# B&R Automation Studio project CControl_Gschneitner (part 3)

#### fbMathTrGutGew.st - Berechnungen des Trockengutes (spez. Gewicht, Wasserentzug, Gewicht Start, Gewicht Ende...)
```iecst
(********************************************************************
 * COPYRIGHT -- LASCO Heu- und Forsttechnik GmbH
 ********************************************************************
 * Library: LascoMath
 * Datei: fbMathTrGutGew.st
 * Autor: Rudolf Lachner
 * Erstellt: 5. März 2014
 ********************************************************************
 * Implementierung der Library LascoMath
 ********************************************************************)

(* Berechnungen des Trockengutes (spez. Gewicht, Wasserentzug, Gewicht Start, Gewicht Ende...) *)
FUNCTION_BLOCK fbMathTrGutGew

	IF (Freigabe = TRUE) THEN

		//Boxentrocknung**************************************************************************************************************************************************
		IF (Anlagentyp = FALSE) THEN

			//Spez. Gewicht des Trockengutes [kg/m³]
			//**************************************

			//Heu
			IF (Trocknungsgut = 0) AND (FeuchteBeiStart <> 0) AND (FeuchteBeiStart < 100) THEN
				TrockengutSpezGewicht		:= (0.0237 * FeuchteBeiStart * FeuchteBeiStart - 0.395 * FeuchteBeiStart + 60.5) * 1.1;
				//Fichte
			ELSIF (Trocknungsgut = 1) AND (FeuchteBeiStart <> 0) AND (FeuchteBeiStart < 100) THEN
				TrockengutSpezGewicht 		:= (0.0313 * FeuchteBeiStart * FeuchteBeiStart + 1.2245 * FeuchteBeiStart + 151.32);
				//Buche
			ELSIF (Trocknungsgut = 2) AND (FeuchteBeiStart <> 0) AND (FeuchteBeiStart < 100) THEN
				TrockengutSpezGewicht 		:= (0.0462 * FeuchteBeiStart * FeuchteBeiStart + 1.7883 * FeuchteBeiStart + 222.47);
				//Mais
			ELSIF (Trocknungsgut = 3) AND (FeuchteBeiStart <> 0) AND (FeuchteBeiStart < 100) THEN
				TrockengutSpezGewicht 		:= (730 + 476 * (FeuchteBeiStart / (100 - FeuchteBeiStart)));
				//Weizen
			ELSIF (Trocknungsgut = 4) AND (FeuchteBeiStart <> 0) AND (FeuchteBeiStart < 100) THEN
				TrockengutSpezGewicht 		:= (680 + 476 * (FeuchteBeiStart / (100 - FeuchteBeiStart)));
			ELSIF (Trocknungsgut = 5) AND (SpezGewichtUser <> 0) AND (FeuchteBeiStart <> 0) AND (FeuchteBeiStart < 100) THEN
				TrockengutSpezGewicht		:= ((SpezGewichtUser - 476) + 476 * (FeuchteBeiStart / (100 - FeuchteBeiStart)));
			ELSE
				TrockengutSpezGewicht		:= CONST_MATH_MAX_VALUE;
			END_IF

			//Trockengut Gewicht bei Trocknungsstart [kg]
			//*******************************************
			IF (TrockengutSpezGewicht <> 0) AND (TrockengutSpezGewicht < CONST_MATH_MAX_VALUE) AND (FuellhoeheTrockengut > 0) AND
				(Boxenflaeche > 0) THEN
				TrockengutGewichtStart		:= Boxenflaeche * FuellhoeheTrockengut * TrockengutSpezGewicht;
			ELSE
				TrockengutGewichtStart		:= 0;
			END_IF

			//Rundballentrocknung***************************************************************************************************************************************************
		ELSE

			//Trockengut Gewicht bei Trocknungsstart [kg]
			//*******************************************
			IF (GewichtProBallen > 0) AND (AnzahlBallen > 0) THEN
				TrockengutGewichtStart		:= GewichtProBallen * AnzahlBallen;
			ELSE
				TrockengutGewichtStart		:= 0;
			END_IF

		END_IF

		//Trockengut Gewicht Substanz [kg]
		//********************************
		IF (TrockengutGewichtStart <> 0) AND (FeuchteBeiStart > 0) THEN
			TrockengutGewichtSubstanz	:= TrockengutGewichtStart - (TrockengutGewichtStart * FeuchteBeiStart / 100);
		ELSE
			TrockengutGewichtSubstanz	:= 0;
		END_IF

		IF (TrockengutGewichtSubstanz < 0) THEN
			TrockengutGewichtSubstanz	:= 0;
		END_IF

		//Trockengut Gewicht Ende [kg]
		//****************************
		IF (TrockengutGewichtSubstanz <> 0) AND (FeuchteEnde > 0) THEN
			loc_TrockengutGewichtEnde	:= ((100 - FeuchteEnde) / 100);
			IF (loc_TrockengutGewichtEnde <> 0) THEN
				TrockengutGewichtEnde	:= TrockengutGewichtSubstanz / loc_TrockengutGewichtEnde;
			ELSE
				TrockengutGewichtEnde	:= 0;
			END_IF
		ELSE
			TrockengutGewichtEnde		:= 0;
		END_IF

		IF (TrockengutGewichtEnde < 0) THEN
			TrockengutGewichtEnde	:= 0;
		END_IF

		//Trockengut Gewicht Wasserentzug [kg]
		//************************************
		IF (TrockengutGewichtStart > 0) AND (TrockengutGewichtEnde > 0) THEN
			TrockengutWasserentzug	:= TrockengutGewichtStart - TrockengutGewichtEnde;
		ELSE
			TrockengutWasserentzug	:= 0;
		END_IF

		//Wasserentzug Seit Start [kg]
		//****************************
		IF (VentilatorInBetrieb) AND (WasserentzugProStunde < CONST_MATH_MAX_VALUE) AND (sekTick) THEN
			WasserentzugSeitStart	:= WasserentzugSeitStart + WasserentzugProStunde / 3600;
		END_IF

		//Aktuelles Trockengut- Gewicht [kg]
		//**********************************
		TrockengutGewichtAktuell	:= TrockengutGewichtStart - WasserentzugSeitStart;

		//Noch abzutrocknendes Wasser [kg]
		//********************************
		RestgewichtWasser			:= TrockengutWasserentzug - WasserentzugSeitStart;

		//Aktuelle Trockengut- Feuchte [%]
		//********************************

		IF (EDGEPOS(CmdKorrekturFeuchte)) THEN
			loc_cmdKorrekturFeuchte	:= TRUE;
		END_IF

		IF TrockengutGewichtEnde > 0 THEN

			//Korrektur durch Bediener ********************************************************************************************************
			IF (FeuchteAktuell <> KorrekturWertFeuchte) AND (EDGEPOS(loc_cmdKorrekturFeuchte)) THEN

				//Check Div0
				temp2		:= (FeuchteEnde - FeuchteBeiStart);
				IF (temp2 = 0) THEN
					temp2	:= temp2 + 0.01;
				END_IF

				temp1 		:= (TrockengutGewichtEnde - TrockengutGewichtStart);
				IF (temp1 = 0) THEN
					temp1	:= temp1 + 0.01;
				END_IF

				//Check Div0
				IF ((KorrekturWertFeuchte - FeuchteBeiStart) = 0) THEN
					KorrekturWertFeuchte	:= KorrekturWertFeuchte + 0.01;
				END_IF

				//Aktuelles Trockengutgewicht neu berechnen
				IF (temp2 <> 0) THEN
					TrockengutGewichtAktuell 	:=  TrockengutGewichtStart + (TrockengutGewichtEnde - TrockengutGewichtStart) / temp2 * (KorrekturWertFeuchte - FeuchteBeiStart);
					WasserentzugSeitStart		:= (TrockengutGewichtStart - TrockengutGewichtAktuell);
				END_IF

				//Check Div0
				IF ((TrockengutGewichtAktuell - TrockengutGewichtStart) = 0) THEN
					TrockengutGewichtAktuell	:= TrockengutGewichtAktuell + 0.01;
				END_IF

				//Aktuelle Trockengut- Feuchte berechnen
				IF (temp1 <> 0) THEN
					FeuchteAktuell := FeuchteBeiStart + (FeuchteEnde - FeuchteBeiStart) / temp1 * (TrockengutGewichtAktuell - TrockengutGewichtStart);
				END_IF

				loc_cmdKorrekturFeuchte		:= FALSE;
				KorrekturWertFeuchte		:= 0.0;

			//Korrektur durch Tabellenprogramm **********************************************************************************************************
			ELSIF (FeuchteAktuell <> KorrekturWertFeuchteRicht) AND (EDGEPOS(CmdKorrekturFeuchteRicht)) THEN

				//Check Div0
				temp1 		:= (TrockengutGewichtEnde - TrockengutGewichtStart);
				IF (temp1 = 0) THEN
					temp1	:= temp1 + 0.01;
				END_IF

				temp2		:= (FeuchteEnde - FeuchteBeiStart);
				IF (temp2 = 0) THEN
					temp2	:= temp2 + 0.01;
				END_IF

				//Check Div0
				IF ((KorrekturWertFeuchteRicht - FeuchteBeiStart) = 0) THEN
					KorrekturWertFeuchteRicht	:= KorrekturWertFeuchteRicht + 0.01;
				END_IF

				//Aktuelles Trockengutgewicht neu berechnen
				IF (temp2 <> 0) THEN
					TrockengutGewichtAktuell 	:= TrockengutGewichtStart + (TrockengutGewichtEnde - TrockengutGewichtStart) / temp2 * (KorrekturWertFeuchteRicht - FeuchteBeiStart);
					WasserentzugSeitStart		:= (TrockengutGewichtStart - TrockengutGewichtAktuell);
				END_IF

				//Check Div0
				IF ((TrockengutGewichtAktuell - TrockengutGewichtStart) = 0) THEN
					TrockengutGewichtAktuell	:= TrockengutGewichtAktuell	+ 0.01;
				END_IF

				//Aktuelle Trockengut- Feuchte berechnen
				IF (temp1 <> 0) THEN
					FeuchteAktuell 	:= FeuchteBeiStart + (FeuchteEnde - FeuchteBeiStart) / temp1 * (TrockengutGewichtAktuell - TrockengutGewichtStart);
				END_IF

				CmdKorrekturFeuchteRicht	:= FALSE;
				KorrekturWertFeuchteRicht	:= 0.0;

			//Automatische Berechnung *******************************************************************************************************************************************************
			ELSIF (KeinStroemungsfuehler = FALSE) THEN

				temp1 := (TrockengutGewichtEnde - TrockengutGewichtStart);
				IF (temp1 = 0) THEN
					temp1	:= temp1 + 0.01;
				END_IF

				//Check Div0
				IF ((TrockengutGewichtAktuell - TrockengutGewichtStart) = 0) THEN
					TrockengutGewichtAktuell	:= TrockengutGewichtAktuell	+ 0.01;
				END_IF

				IF (temp1 <> 0) THEN
					FeuchteAktuell := FeuchteBeiStart + (FeuchteEnde - FeuchteBeiStart) / temp1 * (TrockengutGewichtAktuell - TrockengutGewichtStart);
				END_IF
			END_IF
		ELSE
			FeuchteAktuell	:= 0;
		END_IF

		//Wenn kein Strömungsfühler vorhanden -> Auswertung über Tabellenprogramm
		IF (KeinStroemungsfuehler) AND (Automatikbetrieb) AND (Freigabe)  AND (VentilatorInBetrieb) THEN

			IF (EDGEPOS(Freigabe) OR FeuchteBeiStart <> FeuchteBeiStartMEM) THEN
				firstInit			:= TRUE;
				FeuchteBeiStartMEM	:= FeuchteBeiStart;
			END_IF

			//Richtzeit aktuelle Stufe in Stunden umwandeln
			RichtzeitAktStufeStunden		:= RichtzeitAktStufeTage * 24;

			//Teilung Feuchtigkeit neu berechnen
			IF ((firstInit) OR (CmdKorrekturFeuchteRicht)) AND (RichtzeitAktStufeStunden <> 0) THEN
				TeilungFeuchteRicht			:= FeuchteAktuell / RichtzeitAktStufeStunden;
				firstInit					:= FALSE;
				CmdKorrekturFeuchteRicht	:= FALSE;
			END_IF

			//Mittelwert Feuchteentzug pro Stunde
			IF (stdTick) THEN
				CmdKorrekturFeuchteRicht	:= TRUE;
				KorrekturWertFeuchteRicht	:= FeuchteAktuell - TeilungFeuchteRicht;
			END_IF

		//Kein Automatikbetrieb (oder kein Ventilator in Betrieb)
		ELSIF (KeinStroemungsfuehler) AND (Freigabe) THEN

			//Check Div0
			temp1 := (TrockengutGewichtEnde - TrockengutGewichtStart);
			IF temp1 = 0 THEN
				temp1	:= temp1 + 0.01;
			END_IF

			//Check Div0
			IF ((TrockengutGewichtAktuell - TrockengutGewichtStart) = 0) THEN
				TrockengutGewichtAktuell	:= TrockengutGewichtAktuell	+ 0.01;
			END_IF

			IF (temp1 <> 0) THEN
				FeuchteAktuell := FeuchteBeiStart + (FeuchteEnde - FeuchteBeiStart) / temp1 * (TrockengutGewichtAktuell - TrockengutGewichtStart);
			END_IF

		END_IF

	//keine Freigabe ***************************************************************************************************************************************************************************
	ELSE

		TrockengutSpezGewicht		:= 0;
		TrockengutGewichtStart		:= 0;
		TrockengutGewichtEnde		:= 0;
		TrockengutGewichtSubstanz	:= 0;
		TrockengutWasserentzug		:= 0;
		TrockengutGewichtAktuell	:= 0;
		WasserentzugSeitStart		:= 0;
		loc_TrockengutGewichtEnde	:= 0;

	END_IF

END_FUNCTION_BLOCK
```

#### fbMathTrLftMenge.st - Berechnungen mit Luftmengenmessung
```iecst
(********************************************************************
 * COPYRIGHT -- LASCO Heu- und Forsttechnik GmbH
 ********************************************************************
 * Library: LascoMath
 * Datei: fbMathTrLftMenge.st
 * Autor: Rudolf Lachner
 * Erstellt: 5. März 2014
 ********************************************************************
 * Implementierung der Library LascoMath
 ********************************************************************)

(* Berechnungen mit Luftmengenmessung *)
FUNCTION_BLOCK fbMathTrLftMenge

	IF (Freigabe = TRUE) THEN

		//******************************************************************************************************************************************************************
		//Berechnung Luftmenge Aktuell [m³/h]
		//******************************************************************************************************************************************************************

		//Ventilator 1 + 2 in Betrieb
		IF (Ventilator1Betrieb AND Ventilator2Betrieb AND (DrehzRegelungAktiv OR Ventilator12FixDrehzahl) AND NOT
			ZweiBoxenSystem) THEN

			//Ventilator 2 Manuell -> AUS
			IF (Ventilator2Manuell = TRUE) THEN
				LuftmengeAktuell	:= (Luftgeschw * 3600 * LuftkanalQuerschnitt);
			ELSE
				LuftmengeAktuell	:= (Luftgeschw * 3600 * LuftkanalQuerschnitt) * 2;
			END_IF

			//Ventilator 1 + 2 mit unterschiedlichen Drehzahlen
		ELSIF (Ventilator1Betrieb AND Ventilator2Betrieb AND NOT Ventilator2Manuell AND NOT ZweiBoxenSystem) THEN

			//Drehzahlverhältnis zw. Ventilator 1 und 2 berechnen
			IF (DrehzVent1 > DrehzVent2) THEN
				IF (DrehzVent1 <> 0) THEN
					loc_DrehzVerhaeltnis	:= (1 + DrehzVent2 / DrehzVent1);
				END_IF
			ELSE
				IF (DrehzVent2 <> 0) THEN
					loc_DrehzVerhaeltnis		:= (1 + DrehzVent1 / DrehzVent2);
				END_IF
			END_IF

			LuftmengeAktuell	:= (Luftgeschw * 3600 * LuftkanalQuerschnitt * loc_DrehzVerhaeltnis);

		//Nur Ventilator 1 in Betrieb ODER Zwei-Boxen-System mit 2 Lüftern
		ELSIF (LuftkanalQuerschnitt > 0) AND (Ventilator1Betrieb OR Ventilator2Betrieb) THEN
			LuftmengeAktuell	:= (Luftgeschw * 3600 * LuftkanalQuerschnitt);
		ELSE
			LuftmengeAktuell	:= CONST_MATH_MAX_VALUE;
		END_IF

		//*****************************************************************************************************************************************************************************
		//Berechnung Wasserentzug [kg/h]
		//*****************************************************************************************************************************************************************************

		IF (ZuluftSattDefizit < CONST_MATH_MAX_VALUE) AND (LuftmengeAktuell < CONST_MATH_MAX_VALUE) THEN
			WasserentzugProStunde		:= ((ZuluftSattDefizit * LuftmengeAktuell) / 1000) * OffsetWasserentzug;
		ELSE
			WasserentzugProStunde		:= CONST_MATH_MAX_VALUE;
		END_IF

	ELSE

		LuftmengeAktuell			:= CONST_MATH_MAX_VALUE;
		WasserentzugProStunde		:= CONST_MATH_MAX_VALUE;

	END_IF

END_FUNCTION_BLOCK
```

#### fbMathTrLftDruck.st - Berechnungen mit Drucksensor
```iecst
(********************************************************************
 * COPYRIGHT -- LASCO Heu- und Forsttechnik GmbH
 ********************************************************************
 * Library: LascoMath
 * Datei: fbMathTrLftDruck.st
 * Autor: Rudolf Lachner
 * Erstellt: 5. März 2014
 ********************************************************************
 * Implementierung der Library LascoMath
 ********************************************************************)

(* Berechnungen mit Drucksensor *)
FUNCTION_BLOCK fbMathTrLftDruck

	IF (Freigabe = TRUE) THEN

		LuftDruck_mmWS	:= TrockenluftDruck * 0.102;
		LuftDruck_mbar	:= TrockenluftDruck / 100.0;
		LuftDruck_bar	:= TrockenluftDruck / 100000.0;

	ELSE

		LuftDruck_bar	:= CONST_MATH_MAX_VALUE;
		LuftDruck_mbar	:= CONST_MATH_MAX_VALUE;
		LuftDruck_mmWS	:= CONST_MATH_MAX_VALUE;

	END_IF

END_FUNCTION_BLOCK
```

#### fbMathWetter.st - Auswertung des aktuellen Wetters anhand Rezept und Sättigungsdefizit
```iecst
(********************************************************************
 * COPYRIGHT -- LASCO Heu- und Forsttechnik GmbH
 ********************************************************************
 * Library: LascoMath
 * Datei: fbMathWetter.st
 * Autor: Rudolf Lachner
 * Erstellt: 6. März 2014
 ********************************************************************
 * Implementierung der Library LascoMath
 ********************************************************************)

(* Auswertung des aktuellen Wetters anhand Rezept und Sättigungsdefizit *)
FUNCTION_BLOCK fbMathWetter

	IF (Freigabe = TRUE) THEN

		loc_WetterGut		:= FALSE;
		loc_WetterSchlecht	:= FALSE;

		IF (SattDefizitAktuell >= (SattDefizitRezept + HystereseUmschaltung)) THEN
			loc_WetterGut		:= TRUE;
		ELSIF (SattDefizitAktuell <= (SattDefizitRezept - HystereseUmschaltung)) THEN
			loc_WetterSchlecht	:= TRUE;
		END_IF

		TON_WetterGut.IN		:= loc_WetterGut;
		TON_WetterGut.PT		:= UDINT_TO_TIME(ZeitVerzUmschaltung);
		TON_WetterGut();

		TOF_WetterGut.IN		:= TON_WetterGut.Q;
		TOF_WetterGut.PT		:= UDINT_TO_TIME(ZeitVerzUmschaltung);
		TOF_WetterGut();
		WetterGut				:= TOF_WetterGut.Q;

		TON_WetterSchlecht.IN	:= loc_WetterSchlecht AND NOT WetterGut;
		TON_WetterSchlecht.PT	:= UDINT_TO_TIME(ZeitVerzUmschaltung);
		TON_WetterSchlecht();
		WetterSchlecht			:= TON_WetterSchlecht.Q;

		WetterMittel			:= NOT WetterGut AND NOT WetterSchlecht;

	ELSE

		WetterGut		:= FALSE;
		WetterMittel	:= FALSE;
		WetterSchlecht	:= FALSE;

	END_IF

END_FUNCTION_BLOCK
```

#### fbMathMessblende.st - Berechnungen für Messkanäle mit Messblende
```iecst
(********************************************************************
 * COPYRIGHT --
 ********************************************************************
 * Library: LascoMath
 * Datei: fbMathMessblende.st
 * Autor: rlachner
 * Erstellt: 6. März 2018
 ********************************************************************
 * Implementierung der Library LascoMath
 ********************************************************************)

(* Berechnungen für Messkanäle mit Messblende *)
FUNCTION_BLOCK fbMathMessblende

	IF Enable THEN

		//Volumenstrom aus Luftdichte [AKTUELL]
		//*************************************

		//Luftdichte in Abhängigkeit der Temperatur
		IF (CONST_MATH_GASKONSTANTE * (273 + TemperaturAktuell)) <> 0 THEN
			LuftdichteAktuell	:= CONST_MATH_LUFTDRUCK / (CONST_MATH_GASKONSTANTE * (273 + TemperaturAktuell));
		ELSE
			LuftdichteAktuell	:= CONST_MATH_MAX_VALUE;
		END_IF

		//Luftgeschwindigkeit aus Differenzdruck
		IF (LuftdichteAktuell <> 0) AND (LuftdichteAktuell <> CONST_MATH_MAX_VALUE) THEN
			LuftgeschwindigkeitAktuell	:= CONST_MATH_FAKTOR_DEBIMO * SQRT((2 * DifferenzdruckMessblende) / LuftdichteAktuell);
		ELSE
			LuftgeschwindigkeitAktuell	:= CONST_MATH_MAX_VALUE;
		END_IF

		//Volumenstrom aus Luftgeschwindigkeit
		VolumenstromAktuell := LuftgeschwindigkeitAktuell * Kanalquerschnitt * 3600;

		//Volumenstrom aus Luftdichte [NORM]
		//**********************************

		//Normluftdichte bei 21°C
		LuftdichteNorm	:= CONST_MATH_LUFTDRUCK / (CONST_MATH_GASKONSTANTE * (273 + CONST_MATH_TEMP_NORM));

		//Luftgeschwindigkeit aus Differenzdruck
		LuftgeschwindigkeitNorm		:= CONST_MATH_FAKTOR_DEBIMO * SQRT((2 * DifferenzdruckMessblende) / LuftdichteNorm);

		//Volumenstrom aus Luftgeschwindigkeit
		VolumenstromNorm := LuftgeschwindigkeitNorm * Kanalquerschnitt * 3600;

		//Vergleichsmessung mit Strömungsfühler
		VolumenstromVergleich	:= LuftgeschwindigkeitSensor * Kanalquerschnitt * 3600;

	ELSE

		LuftdichteAktuell			:= 0.0;
		LuftdichteNorm				:= 0.0;
		LuftgeschwindigkeitAktuell	:= 0.0;
		LuftgeschwindigkeitNorm		:= 0.0;
		VolumenstromAktuell			:= 0.0;
		VolumenstromNorm			:= 0.0;
		VolumenstromVergleich		:= 0.0;

	END_IF

END_FUNCTION_BLOCK
```

### Library Logical/Libraries/LascoReg (IEC, version 1.00.0) - Lasco Regler

#### LascoReg.var - Exportierte Konstanten
```iecst
(********************************************************************
 * COPYRIGHT -- LASCO Heu- und Forsttechnik GmbH
 ********************************************************************
 * Library: LascoReg
 * Datei: LascoReg.var
 * Autor: Rudolf Lachner
 * Erstellt: 16. Juli 2014
 ********************************************************************
 * Konstanten der Library LascoReg
 ********************************************************************)
VAR CONSTANT
	FBREG_MODUS_AUS : USINT := 0;
	FBREG_MODUS_AUTO : USINT := 1;
	FBREG_MODUS_MANUELL : USINT := 102;
	FBREG_MODUS_OPEN : USINT := 103;
	FBREG_MODUS_CLOSE : USINT := 104;
	FBREG_MODUS_FREEZE : USINT := 105;
END_VAR
```

#### LascoReg.fun - Exportierte Funktionen und Funktionsblöcke
```iecst
(********************************************************************
 * COPYRIGHT -- LASCO Heu- und Forsttechnik GmbH
 ********************************************************************
 * Library: LascoReg
 * Datei: LascoReg.fun
 * Autor: Rudolf Lachner
 * Erstellt: 16. Juli 2014
 ********************************************************************
 * Funktionen und Funktionsblöcke der Library LascoReg
 ********************************************************************)

FUNCTION_BLOCK fbRegPidReglerAllg (*Standard- PID- Regler*) (*$GROUP=Anwender*)
	VAR_INPUT
		Freigabe : BOOL;
		Hysterese : REAL;
		RampeMax : REAL;
		Invert : BOOL;
		WindupDaempfung : REAL;
		P_Anteil : REAL;
		AbschwaechungSollwert : REAL;
		D_Filterzeit : REAL;
		I_Anteil : REAL;
		D_Anteil : REAL;
		Aufschaltgroesse : REAL;
		Hold_I : BOOL;
		Mode : USINT;
		Sollwert : REAL;
		Istwert : REAL;
		StellgroesseManuell : REAL;
		StellgroesseMin : REAL;
		StellgroesseMax : REAL;
		RegelbereichMin : REAL;
		Fehlerverzoegerung : UDINT;
		RegelbereichMax : REAL;
	END_VAR
	VAR_OUTPUT
		Stellgroesse : REAL;
		Regelabweichung : REAL;
		FehlerRegelbereichMin : BOOL;
		FehlerRegelbereichMax : BOOL;
		WarnungRegelbereichMin : BOOL;
		WarnungRegelbereichMax : BOOL;
	END_VAR
	VAR
		PID_Para : LCRPIDpara;
		PID : LCRPID;
		TON_FehlerverzoegerungMin : TON;
		TON_FehlerverzoegerungMax : TON;
	END_VAR
	VAR_INPUT
		QuitFehler : BOOL;
	END_VAR
	VAR
		LCRLimScal_0 : LCRLimScal;
	END_VAR
END_FUNCTION_BLOCK
```

#### fbRegPidReglerAllg.st - Standard- PID- Regler
```iecst
(********************************************************************
 * COPYRIGHT -- LASCO Heu- und Forsttechnik GmbH
 ********************************************************************
 * Library: LascoReg
 * Datei: fbRegPidReglerAllg.st
 * Autor: Rudolf Lachner
 * Erstellt: 16. Juli 2014
 ********************************************************************
 * Implementierung der Library LascoReg
 ********************************************************************)

(* Standard- PID- Regler *)
FUNCTION_BLOCK fbRegPidReglerAllg

	IF (Freigabe) THEN

		//Parametrierungsbaustein des Reglers
		PID_Para.enable			:= Freigabe;
		PID_Para.enter			:= Freigabe;
		PID_Para.deadband		:= Hysterese;
		PID_Para.deadband_mode	:= LCRPID_DEADBAND_MODE_STANDARD;
		PID_Para.dY_max			:= RampeMax;
		PID_Para.d_mode			:= LCRPID_D_MODE_E;
		PID_Para.fbk_mode		:= LCRPID_FBK_MODE_INTERN;
		PID_Para.invert			:= Invert;
		PID_Para.Kfbk			:= WindupDaempfung;
		PID_Para.Kp				:= P_Anteil;
		PID_Para.Kw				:= AbschwaechungSollwert;
		PID_Para.Tf				:= D_Filterzeit;
		PID_Para.Tn				:= I_Anteil;
		PID_Para.Tv				:= D_Anteil;
		PID_Para.WX_min			:= 0.0;
		PID_Para.WX_max			:= 100.0;

		//PID- Reglerbaustein
		PID.enable				:= Freigabe;
		PID.A					:= Aufschaltgroesse;
		PID.hold_I				:= Hold_I;
		PID.ident				:= PID_Para.ident;
		PID.mode				:= Mode;
		PID.W					:= Sollwert;
		PID.X					:= Istwert;
		PID.Y_fbk				:= 0.0;
		PID.Y_man				:= StellgroesseManuell;
		PID.Y_min				:= 0.0;
		PID.Y_max				:= 100.0;

		//Min-Max des Reglers von 0-100% auf Stellgröße skalieren
		LCRLimScal_0(x := PID.Y, x1 := 0, y1 := StellgroesseMin, x2 := 100, y2 := StellgroesseMax);

		Stellgroesse			:= LCRLimScal_0.y;
		Regelabweichung			:= PID.e;

		//Warnungs- und Fehlergenerierung bei Erreichen des Min/Max- Regelbereiches
		TON_FehlerverzoegerungMin.IN	:= (Istwert < RegelbereichMin) AND Freigabe AND NOT QuitFehler;
		TON_FehlerverzoegerungMin.PT	:= UDINT_TO_TIME(Fehlerverzoegerung);

		TON_FehlerverzoegerungMax.IN	:= (Istwert > RegelbereichMax) AND Freigabe AND NOT QuitFehler;
		TON_FehlerverzoegerungMax.PT	:= UDINT_TO_TIME(Fehlerverzoegerung);

		WarnungRegelbereichMin			:= TON_FehlerverzoegerungMin.IN;
		WarnungRegelbereichMax			:= TON_FehlerverzoegerungMax.IN;

		FehlerRegelbereichMin			:= TON_FehlerverzoegerungMin.Q;
		FehlerRegelbereichMax			:= TON_FehlerverzoegerungMax.Q;

		//Funktionsbausteine aufrufen
		PID_Para();
		PID();
		TON_FehlerverzoegerungMax();
		TON_FehlerverzoegerungMin();

	ELSE

		Stellgroesse			:= 0.0;
		Regelabweichung			:= 0.0;
		WarnungRegelbereichMax	:= FALSE;
		WarnungRegelbereichMin	:= FALSE;
		FehlerRegelbereichMax	:= FALSE;
		FehlerRegelbereichMin	:= FALSE;

	END_IF

END_FUNCTION_BLOCK
```

### Library Logical/Libraries/LascoTrock (IEC, version 1.00.0) - Funktionsblöcke für Trocknungsanlagen

#### LascoTrock.typ - Exportierte Datentypen
```iecst
(********************************************************************
 * COPYRIGHT -- LASCO Heu- und Forsttechik GmbH
 ********************************************************************
 * Library: LascoTrock
 * Datei: LascoTrock.typ
 * Autor: Rudolf Lachner
 * Erstellt: 10. März 2014
 ********************************************************************
 * Datentypen der Library LascoTrock
 ********************************************************************)

TYPE
	enumStepTrockVent :
		(
		WARTEN_FBTROCK := 0,
		VENT_EIN_FBTROCK := 1,
		VENT_AUS_FBTROCK := 2,
		KLAPPEN_AUF_FBTROCK := 3,
		KLAPPEN_ZU_FBTROCK := 4,
		LA_EIN_VORBEREITUNG_FBTROCK := 5,
		LA_EIN_FBTROCK := 6,
		LA_AUS_VORBEREITUNG_FBTROCK := 7,
		MESSUNG_FBTROCK := 8,
		TARIFABSCHALTUNG_FBTROCK := 9
		);
END_TYPE
```

#### LascoTrock.var - Exportierte Konstanten
```iecst
(********************************************************************
 * COPYRIGHT -- LASCO Heu- und Forsttechnik GmbH
 ********************************************************************
 * Library: LascoTrock
 * Datei: LascoTrock.var
 * Autor: Rudolf Lachner
 * Erstellt: 10. März 2014
 ********************************************************************
 * Konstanten der Library LascoTrock
 ********************************************************************)
VAR CONSTANT
	TROCK_VARIANTEN_NAMEN1 : ARRAY[0..120] OF STRING[100] := ['Keine gültige Variante','1 Ventilator','1 Ventilator, 2 Boxen','1 Ventilator, Betriebsmeldung SHO','1 Ventilator, Betriebsmeldung SHO, 2 Boxen','1 Ventilator, Betriebsmeldung SHO, BSK','1 Ventilator, Betriebsmeldung SHO, BSK, 2 Boxen','1 Ventilator, Betriebsmeldung WLO','1 Ventilator, Betriebsmeldung WLO, 2 Boxen','1 Ventilator, Betriebsmeldung WLO, BSK','1 Ventilator, Betriebsmeldung WLO, BSK, 2 Boxen','1 Ventilator, Betriebsmeldung WLO und SHO','1 Ventilator, Betriebsmeldung WLO und SHO, 2 Boxen','1 Ventilator, Betriebsmeldung WLO und SHO, BSK','1 Ventilator, Betriebsmeldung WLO und SHO, BSK, 2 Boxen','1 Ventilator, WLO','1 Ventilator, WLO, 2 Boxen','1 Ventilator, WLO, BSK','1 Ventilator, WLO, BSK, 2 Boxen','1 Ventilator, WLO, Betriebsmeldung SHO','1 Ventilator, WLO, Betriebsmeldung SHO, 2 Boxen','1 Ventilator, WLO, Betriebsmeldung SHO, BSK','1 Ventilator, WLO, Betriebsmeldung SHO, BSK, 2 Boxen','1 Ventilator, WLO, Betriebsmeldung WLO','1 Ventilator, WLO, Betriebsmeldung WLO, 2 Boxen','1 Ventilator, WLO, Betriebsmeldung WLO, BSK','1 Ventilator, WLO, Betriebsmeldung WLO, BSK, 2 Boxen','1 Ventilator, WLO, Betriebsmeldung WLO und SHO','1 Ventilator, WLO, Betriebsmeldung WLO und SHO, 2 Boxen','1 Ventilator, WLO, Betriebsmeldung WLO und SHO, BSK','1 Ventilator, WLO, Betriebsmeldung WLO und SHO, BSK, 2 Boxen','1 Ventilator, LE','1 Ventilator, LE, 2 Boxen','1 Ventilator, LE, Betriebsmeldung SHO','1 Ventilator, LE, Betriebsmeldung SHO, 2 Boxen','1 Ventilator, LE, Betriebsmeldung SHO, BSK','1 Ventilator, LE, Betriebsmeldung SHO, BSK, 2 Boxen','1 Ventilator, LE, Betriebsmeldung WLO','1 Ventilator, LE, Betriebsmeldung WLO, 2 Boxen','1 Ventilator, LE, Betriebsmeldung WLO, BSK','1 Ventilator, LE, Betriebsmeldung WLO, BSK, 2 Boxen','1 Ventilator, LE, Betriebsmeldung WLO und SHO','1 Ventilator, LE, Betriebsmeldung WLO und SHO, 2 Boxen','1 Ventilator, LE, Betriebsmeldung WLO und SHO, BSK','1 Ventilator, LE, Betriebsmeldung WLO und SHO, BSK, 2 Boxen','1 Ventilator, LE, WLO','1 Ventilator, LE, WLO, 2 Boxen','1 Ventilator, LE, WLO, BSK','1 Ventilator, LE, WLO, BSK, 2 Boxen','1 Ventilator, LE, WLO, Betriebsmeldung SHO','1 Ventilator, LE, WLO, Betriebsmeldung SHO, 2 Boxen','1 Ventilator, LE, WLO, Betriebsmeldung SHO, BSK','1 Ventilator, LE, WLO, Betriebsmeldung SHO, BSK, 2 Boxen','1 Ventilator, LE, WLO, Betriebsmeldung WLO','1 Ventilator, LE, WLO, Betriebsmeldung WLO, 2 Boxen','1 Ventilator, LE, WLO, Betriebsmeldung WLO, BSK','1 Ventilator, LE, WLO, Betriebsmeldung WLO, BSK, 2 Boxen','1 Ventilator, LE, WLO, Betriebsmeldung WLO und SHO','1 Ventilator, LE, WLO, Betriebsmeldung WLO und SHO, 2 Boxen','1 Ventilator, LE, WLO, Betriebsmeldung WLO und SHO, BSK','1 Ventilator, LE, WLO, Betriebsmeldung WLO und SHO, BSK, 2 Boxen','2 Ventilatoren','2 Ventilatoren, 2 Boxen','2 Ventilatoren, Betriebsmeldung SHO','2 Ventilatoren, Betriebsmeldung SHO, 2 Boxen','2 Ventilatoren, Betriebsmeldung SHO, BSK','2 Ventilatoren, Betriebsmeldung SHO, BSK, 2 Boxen','2 Ventilatoren, Betriebsmeldung WLO','2 Ventilatoren, Betriebsmeldung WLO, 2 Boxen','2 Ventilatoren, Betriebsmeldung WLO, BSK','2 Ventilatoren, Betriebsmeldung WLO, BSK, 2 Boxen','2 Ventilatoren, Betriebsmeldung WLO und SHO','2 Ventilatoren, Betriebsmeldung WLO und SHO, 2 Boxen','2 Ventilatoren, Betriebsmeldung WLO und SHO, BSK','2 Ventilatoren, Betriebsmeldung WLO und SHO, BSK, 2 Boxen','2 Ventilatoren, WLO','2 Ventilatoren, WLO, 2 Boxen','2 Ventilatoren, WLO, BSK','2 Ventilatoren, WLO, BSK, 2 Boxen','2 Ventilatoren, WLO, Betriebsmeldung SHO','2 Ventilatoren, WLO, Betriebsmeldung SHO, 2 Boxen','2 Ventilatoren, WLO, Betriebsmeldung SHO, BSK','2 Ventilatoren, WLO, Betriebsmeldung SHO, BSK, 2 Boxen','2 Ventilatoren, WLO, Betriebsmeldung WLO','2 Ventilatoren, WLO, Betriebsmeldung WLO, 2 Boxen','2 Ventilatoren, WLO, Betriebsmeldung WLO, BSK','2 Ventilatoren, WLO, Betriebsmeldung WLO, BSK, 2 Boxen','2 Ventilatoren, WLO, Betriebsmeldung WLO und SHO','2 Ventilatoren, WLO, Betriebsmeldung WLO und SHO, 2 Boxen','2 Ventilatoren, WLO, Betriebsmeldung WLO und SHO, BSK','2 Ventilatoren, WLO, Betriebsmeldung WLO und SHO, BSK, 2 Boxen','2 Ventilatoren, LE','2 Ventilatoren, LE, 2 Boxen','2 Ventilatoren, LE, Betriebsmeldung SHO','2 Ventilatoren, LE, Betriebsmeldung SHO, 2 Boxen','2 Ventilatoren, LE, Betriebsmeldung SHO, BSK','2 Ventilatoren, LE, Betriebsmeldung SHO, BSK, 2 Boxen','2 Ventilatoren, LE, Betriebsmeldung WLO','2 Ventilatoren, LE, Betriebsmeldung WLO, 2 Boxen','2 Ventilatoren, LE, Betriebsmeldung WLO, BSK','2 Ventilatoren, LE, Betriebsmeldung WLO, BSK, 2 Boxen','2 Ventilatoren, LE, Betriebsmeldung WLO und SHO','2 Ventilatoren, LE, Betriebsmeldung WLO und SHO, 2 Boxen','2 Ventilatoren, LE, Betriebsmeldung WLO und SHO, BSK','2 Ventilatoren, LE, Betriebsmeldung WLO und SHO, BSK, 2 Boxen','2 Ventilatoren, LE, WLO','2 Ventilatoren, LE, WLO, 2 Boxen','2 Ventilatoren, LE, WLO, BSK','2 Ventilatoren, LE, WLO, BSK, 2 Boxen','2 Ventilatoren, LE, WLO, Betriebsmeldung SHO','2 Ventilatoren, LE, WLO, Betriebsmeldung SHO, 2 Boxen','2 Ventilatoren, LE, WLO, Betriebsmeldung SHO, BSK','2 Ventilatoren, LE, WLO, Betriebsmeldung SHO, BSK, 2 Boxen','2 Ventilatoren, LE, WLO, Betriebsmeldung WLO','2 Ventilatoren, LE, WLO, Betriebsmeldung WLO, 2 Boxen','2 Ventilatoren, LE, WLO, Betriebsmeldung WLO, BSK','2 Ventilatoren, LE, WLO, Betriebsmeldung WLO, BSK, 2 Boxen','2 Ventilatoren, LE, WLO, Betriebsmeldung WLO und SHO','2 Ventilatoren, LE, WLO, Betriebsmeldung WLO und SHO, 2 Boxen','2 Ventilatoren, LE, WLO, Betriebsmeldung WLO und SHO, BSK','2 Ventilatoren, LE, WLO, Betriebsmeldung WLO und SHO, BSK, 2 Boxen'];
	TROCK_VARIANTEN_NAMEN : ARRAY[0..120] OF STRING[100] := ['Keine gültige Variante','1 Ventilator','1 Ventilator, 2 Boxen','1 Ventilator, Betriebsmeldung SHO','1 Ventilator, Betriebsmeldung SHO, 2 Boxen','1 Ventilator, Betriebsmeldung SHO, BSK','1 Ventilator, Betriebsmeldung SHO, BSK, 2 Boxen','1 Ventilator, Betriebsmeldung WLO','1 Ventilator, Betriebsmeldung WLO, 2 Boxen','1 Ventilator, Betriebsmeldung WLO, BSK','1 Ventilator, Betriebsmeldung WLO, BSK, 2 Boxen','1 Ventilator, Betriebsmeldung WLO und SHO','1 Ventilator, Betriebsmeldung WLO und SHO, 2 Boxen','1 Ventilator, Betriebsmeldung WLO und SHO, BSK','1 Ventilator, Betriebsmeldung WLO und SHO, BSK, 2 Boxen','1 Ventilator, WLO','1 Ventilator, WLO, 2 Boxen','1 Ventilator, WLO, BSK','1 Ventilator, WLO, BSK, 2 Boxen','1 Ventilator, WLO, Betriebsmeldung SHO','1 Ventilator, WLO, Betriebsmeldung SHO, 2 Boxen','1 Ventilator, WLO, Betriebsmeldung SHO, BSK','1 Ventilator, WLO, Betriebsmeldung SHO, BSK, 2 Boxen','1 Ventilator, WLO, Betriebsmeldung WLO','1 Ventilator, WLO, Betriebsmeldung WLO, 2 Boxen','1 Ventilator, WLO, Betriebsmeldung WLO, BSK','1 Ventilator, WLO, Betriebsmeldung WLO, BSK, 2 Boxen','1 Ventilator, WLO, Betriebsmeldung WLO und SHO','1 Ventilator, WLO, Betriebsmeldung WLO und SHO, 2 Boxen','1 Ventilator, WLO, Betriebsmeldung WLO und SHO, BSK','1 Ventilator, WLO, Betriebsmeldung WLO und SHO, BSK, 2 Boxen','1 Ventilator, LE','1 Ventilator, LE, 2 Boxen','1 Ventilator, LE, Betriebsmeldung SHO','1 Ventilator, LE, Betriebsmeldung SHO, 2 Boxen','1 Ventilator, LE, Betriebsmeldung SHO, BSK','1 Ventilator, LE, Betriebsmeldung SHO, BSK, 2 Boxen','1 Ventilator, LE, Betriebsmeldung WLO','1 Ventilator, LE, Betriebsmeldung WLO, 2 Boxen','1 Ventilator, LE, Betriebsmeldung WLO, BSK','1 Ventilator, LE, Betriebsmeldung WLO, BSK, 2 Boxen','1 Ventilator, LE, Betriebsmeldung WLO und SHO','1 Ventilator, LE, Betriebsmeldung WLO und SHO, 2 Boxen','1 Ventilator, LE, Betriebsmeldung WLO und SHO, BSK','1 Ventilator, LE, Betriebsmeldung WLO und SHO, BSK, 2 Boxen','1 Ventilator, LE, WLO','1 Ventilator, LE, WLO, 2 Boxen','1 Ventilator, LE, WLO, BSK','1 Ventilator, LE, WLO, BSK, 2 Boxen','1 Ventilator, LE, WLO, Betriebsmeldung SHO','1 Ventilator, LE, WLO, Betriebsmeldung SHO, 2 Boxen','1 Ventilator, LE, WLO, Betriebsmeldung SHO, BSK','1 Ventilator, LE, WLO, Betriebsmeldung SHO, BSK, 2 Boxen','1 Ventilator, LE, WLO, Betriebsmeldung WLO','1 Ventilator, LE, WLO, Betriebsmeldung WLO, 2 Boxen','1 Ventilator, LE, WLO, Betriebsmeldung WLO, BSK','1 Ventilator, LE, WLO, Betriebsmeldung WLO, BSK, 2 Boxen','1 Ventilator, LE, WLO, Betriebsmeldung WLO und SHO','1 Ventilator, LE, WLO, Betriebsmeldung WLO und SHO, 2 Boxen','1 Ventilator, LE, WLO, Betriebsmeldung WLO und SHO, BSK','1 Ventilator, LE, WLO, Betriebsmeldung WLO und SHO, BSK, 2 Boxen','2 Ventilatoren','2 Ventilatoren, 2 Boxen','2 Ventilatoren, Betriebsmeldung SHO','2 Ventilatoren, Betriebsmeldung SHO, 2 Boxen','2 Ventilatoren, Betriebsmeldung SHO, BSK','2 Ventilatoren, Betriebsmeldung SHO, BSK, 2 Boxen','2 Ventilatoren, Betriebsmeldung WLO','2 Ventilatoren, Betriebsmeldung WLO, 2 Boxen','2 Ventilatoren, Betriebsmeldung WLO, BSK','2 Ventilatoren, Betriebsmeldung WLO, BSK, 2 Boxen','2 Ventilatoren, Betriebsmeldung WLO und SHO','2 Ventilatoren, Betriebsmeldung WLO und SHO, 2 Boxen','2 Ventilatoren, Betriebsmeldung WLO und SHO, BSK','2 Ventilatoren, Betriebsmeldung WLO und SHO, BSK, 2 Boxen','2 Ventilatoren, WLO','2 Ventilatoren, WLO, 2 Boxen','2 Ventilatoren, WLO, BSK','2 Ventilatoren, WLO, BSK, 2 Boxen','2 Ventilatoren, WLO, Betriebsmeldung SHO','2 Ventilatoren, WLO, Betriebsmeldung SHO, 2 Boxen','2 Ventilatoren, WLO, Betriebsmeldung SHO, BSK','2 Ventilatoren, WLO, Betriebsmeldung SHO, BSK, 2 Boxen','2 Ventilatoren, WLO, Betriebsmeldung WLO','2 Ventilatoren, WLO, Betriebsmeldung WLO, 2 Boxen','2 Ventilatoren, WLO, Betriebsmeldung WLO, BSK','2 Ventilatoren, WLO, Betriebsmeldung WLO, BSK, 2 Boxen','2 Ventilatoren, WLO, Betriebsmeldung WLO und SHO','2 Ventilatoren, WLO, Betriebsmeldung WLO und SHO, 2 Boxen','2 Ventilatoren, WLO, Betriebsmeldung WLO und SHO, BSK','2 Ventilatoren, WLO, Betriebsmeldung WLO und SHO, BSK, 2 Boxen','2 Ventilatoren, LE','2 Ventilatoren, LE, 2 Boxen','2 Ventilatoren, LE, Betriebsmeldung SHO','2 Ventilatoren, LE, Betriebsmeldung SHO, 2 Boxen','2 Ventilatoren, LE, Betriebsmeldung SHO, BSK','2 Ventilatoren, LE, Betriebsmeldung SHO, BSK, 2 Boxen','2 Ventilatoren, LE, Betriebsmeldung WLO','2 Ventilatoren, LE, Betriebsmeldung WLO, 2 Boxen','2 Ventilatoren, LE, Betriebsmeldung WLO, BSK','2 Ventilatoren, LE, Betriebsmeldung WLO, BSK, 2 Boxen','2 Ventilatoren, LE, Betriebsmeldung WLO und SHO','2 Ventilatoren, LE, Betriebsmeldung WLO und SHO, 2 Boxen','2 Ventilatoren, LE, Betriebsmeldung WLO und SHO, BSK','2 Ventilatoren, LE, Betriebsmeldung WLO und SHO, BSK, 2 Boxen','2 Ventilatoren, LE, WLO','2 Ventilatoren, LE, WLO, 2 Boxen','2 Ventilatoren, LE, WLO, BSK','2 Ventilatoren, LE, WLO, BSK, 2 Boxen','2 Ventilatoren, LE, WLO, Betriebsmeldung SHO','2 Ventilatoren, LE, WLO, Betriebsmeldung SHO, 2 Boxen','2 Ventilatoren, LE, WLO, Betriebsmeldung SHO, BSK','2 Ventilatoren, LE, WLO, Betriebsmeldung SHO, BSK, 2 Boxen','2 Ventilatoren, LE, WLO, Betriebsmeldung WLO','2 Ventilatoren, LE, WLO, Betriebsmeldung WLO, 2 Boxen','2 Ventilatoren, LE, WLO, Betriebsmeldung WLO, BSK','2 Ventilatoren, LE, WLO, Betriebsmeldung WLO, BSK, 2 Boxen','2 Ventilatoren, LE, WLO, Betriebsmeldung WLO und SHO','2 Ventilatoren, LE, WLO, Betriebsmeldung WLO und SHO, 2 Boxen','2 Ventilatoren, LE, WLO, Betriebsmeldung WLO und SHO, BSK','2 Ventilatoren, LE, WLO, Betriebsmeldung WLO und SHO, BSK, 2 Boxen'];
END_VAR
```

#### LascoTrock.fun - Exportierte Funktionen und Funktionsblöcke
```iecst
(********************************************************************
 * COPYRIGHT -- LASCO Heu- und Forsttechnik GmbH
 ********************************************************************
 * Library: LascoTrock
 * Datei: LascoTrock.fun
 * Autor: Rudolf Lachner
 * Erstellt: 10. März 2014
 ********************************************************************
 * Funktionen und Funktionsblöcke der Library LascoTrock
 ********************************************************************)

FUNCTION_BLOCK fbTrockZeitprogramm (*Generierung von Start- und Stoppsignalen aus Zeitprogramm*) (*$GROUP=Anwender*)
	VAR_INPUT
		Freigabe : BOOL; (*Freigabe des Funktionsblockes*)
		AktZeit : REAL; (*Aktuelle Zeit im Format hhmm*)
		StartZeit1 : REAL; (*Startzeit 1*)
		StartZeit2 : REAL; (*Startzeit 2*)
		StartZeit3 : REAL; (*Startzeit 3*)
		StartZeit4 : REAL; (*Startzeit 4*)
		StartZeit5 : REAL; (*Startzeit 5*)
		StoppZeit1 : REAL; (*Stoppzeit 1*)
		StoppZeit2 : REAL; (*Stoppzeit 2*)
		StoppZeit3 : REAL; (*Stoppzeit 3*)
		StoppZeit4 : REAL; (*Stoppzeit 4*)
		StoppZeit5 : REAL; (*Stoppzeit 5*)
	END_VAR
	VAR_OUTPUT
		FreigabeZeitprogramm : BOOL; (*Freigabe von Zeitprogramm*)
	END_VAR
	VAR
		FreigZeitfenster1 : BOOL;
		FreigZeitfenster2 : BOOL;
		FreigZeitfenster3 : BOOL;
		FreigZeitfenster4 : BOOL;
		FreigZeitfenster5 : BOOL;
	END_VAR
END_FUNCTION_BLOCK

FUNCTION_BLOCK fbTrockLaufPause (*Lauf- und Pausenprogramm*) (*$GROUP=Anwender*)
	VAR_INPUT
		Freigabe : BOOL;
		ZeitLauf : UDINT; (*Laufzeit*)
		ZeitLaufMin : UDINT; (*Mindestlaufzeit*)
		Tick : BOOL; (*Zeittick*)
		Reset : BOOL; (*Reset*)
		ZeitPause : UDINT;
	END_VAR
	VAR_OUTPUT
		FreigabeLpPrg : BOOL; (*Freigabe von Lauf/Pausenprogramm*)
		RestzeitPause : UDINT;
		RestzeitLauf : UDINT;
	END_VAR
	VAR
		currStep : USINT;
		nextStep : USINT;
		CounterLauf : UDINT;
		CounterPause : UDINT;
		zzEdge00000 : BOOL;
		zzEdge00001 : BOOL;
	END_VAR
END_FUNCTION_BLOCK

{REDUND_UNREPLICABLE} FUNCTION_BLOCK fbTrockNachtrock (*Funktionsbaustein Nachtrocknung*) (*$GROUP=Anwender*)
	VAR_INPUT
		Freigabe : {REDUND_UNREPLICABLE} BOOL;
		AktZeit : {REDUND_UNREPLICABLE} REAL;
		StartZeit1 : {REDUND_UNREPLICABLE} REAL;
		StartZeit2 : {REDUND_UNREPLICABLE} REAL;
		StartZeit3 : {REDUND_UNREPLICABLE} REAL;
		StoppZeit1 : {REDUND_UNREPLICABLE} REAL;
		StoppZeit2 : {REDUND_UNREPLICABLE} REAL;
		StoppZeit3 : {REDUND_UNREPLICABLE} REAL;
		TagTick : {REDUND_UNREPLICABLE} BOOL;
		ZyklusTageSoll : {REDUND_UNREPLICABLE} UDINT;
		DauerNachtrocknungTage : {REDUND_UNREPLICABLE} UDINT;
		StdTick : {REDUND_UNREPLICABLE} BOOL;
	END_VAR
	VAR_OUTPUT
		FreigabeNachtrocknung : {REDUND_UNREPLICABLE} BOOL;
		TageNachtrocknungAktiv : {REDUND_UNREPLICABLE} UDINT;
		ZyklusTageIst : {REDUND_UNREPLICABLE} UDINT;
		AktTagFreigabe : {REDUND_UNREPLICABLE} BOOL;
		NachtrocknungFertig : {REDUND_UNREPLICABLE} BOOL;
		StdNachtrocknung : {REDUND_UNREPLICABLE} UDINT;
	END_VAR
	VAR
		FreigZeitfenster1 : {REDUND_UNREPLICABLE} BOOL;
		FreigZeitfenster2 : {REDUND_UNREPLICABLE} BOOL;
		FreigZeitfenster3 : {REDUND_UNREPLICABLE} BOOL;
	END_VAR
END_FUNCTION_BLOCK

{REDUND_UNREPLICABLE} FUNCTION_BLOCK fbTrockTarifabsch (*Funktionsbaustein Tarifabschaltung*) (*$GROUP=Anwender*)
	VAR_INPUT
		Freigabe : {REDUND_UNREPLICABLE} BOOL;
		StartMin1 : {REDUND_UNREPLICABLE} REAL;
		StartStd1 : {REDUND_UNREPLICABLE} REAL;
		StartMin2 : {REDUND_UNREPLICABLE} REAL;
		StartStd2 : {REDUND_UNREPLICABLE} REAL;
		StartMin3 : {REDUND_UNREPLICABLE} REAL;
		StartStd3 : {REDUND_UNREPLICABLE} REAL;
		AktZeit : {REDUND_UNREPLICABLE} REAL;
		StoppMin1 : {REDUND_UNREPLICABLE} REAL;
		StoppStd1 : {REDUND_UNREPLICABLE} REAL;
		StoppMin2 : {REDUND_UNREPLICABLE} REAL;
		StoppStd2 : {REDUND_UNREPLICABLE} REAL;
		StoppMin3 : {REDUND_UNREPLICABLE} REAL;
		StoppStd3 : {REDUND_UNREPLICABLE} REAL;
		VorlaufzeitLuftaufbMin : {REDUND_UNREPLICABLE} REAL;
	END_VAR
	VAR_OUTPUT
		TarifabschaltungLuftaufbEin : {REDUND_UNREPLICABLE} BOOL;
		TarifabschaltungEin : {REDUND_UNREPLICABLE} BOOL;
	END_VAR
	VAR
		FreigZeitfenster1 : {REDUND_UNREPLICABLE} BOOL;
		FreigZeitfenster2 : {REDUND_UNREPLICABLE} BOOL;
		FreigZeitfenster3 : {REDUND_UNREPLICABLE} BOOL;
		FreigabeZeitfensterLuftaufb1 : {REDUND_UNREPLICABLE} BOOL;
		FreigabeZeitfensterLuftaufb2 : {REDUND_UNREPLICABLE} BOOL;
		FreigabeZeitfensterLuftaufb3 : {REDUND_UNREPLICABLE} BOOL;
		StartZeit2 : {REDUND_UNREPLICABLE} REAL;
		StartZeit3 : {REDUND_UNREPLICABLE} REAL;
		StartZeit1 : {REDUND_UNREPLICABLE} REAL;
		StoppZeit2 : {REDUND_UNREPLICABLE} REAL;
		StoppZeit3 : {REDUND_UNREPLICABLE} REAL;
		StoppZeit1 : {REDUND_UNREPLICABLE} REAL;
		loc_StdVorlaufzeitREAL : {REDUND_UNREPLICABLE} REAL;
		loc_StdVorlaufzeit : {REDUND_UNREPLICABLE} INT;
		loc_MinVorlaufzeit : {REDUND_UNREPLICABLE} REAL;
		loc_ZwischenergStartStd : {REDUND_UNREPLICABLE} REAL;
		loc_StartStdLuftaufb : {REDUND_UNREPLICABLE} REAL;
		loc_ZwischenergStartMin : {REDUND_UNREPLICABLE} REAL;
		loc_StartMinLuftaufb : {REDUND_UNREPLICABLE} REAL;
		StartZeitLuftaufb1 : {REDUND_UNREPLICABLE} REAL;
		StartZeitLuftaufb2 : {REDUND_UNREPLICABLE} REAL;
		StartZeitLuftaufb3 : {REDUND_UNREPLICABLE} REAL;
	END_VAR
END_FUNCTION_BLOCK

{REDUND_UNREPLICABLE} FUNCTION_BLOCK fbTrockStrombegr (*Strombegrenzung in bestimmten Zeitfenstern*) (*$GROUP=Anwender*)
	VAR_INPUT
		Freigabe : {REDUND_UNREPLICABLE} BOOL;
		StartZeit1 : {REDUND_UNREPLICABLE} REAL;
		StoppZeit1 : {REDUND_UNREPLICABLE} REAL;
		AktZeit : {REDUND_UNREPLICABLE} REAL;
		StartZeit2 : {REDUND_UNREPLICABLE} REAL;
		StoppZeit2 : {REDUND_UNREPLICABLE} REAL;
		StartZeit3 : {REDUND_UNREPLICABLE} REAL;
		StoppZeit3 : {REDUND_UNREPLICABLE} REAL;
		DrehzahlBegrenzung1 : {REDUND_UNREPLICABLE} REAL;
		DrehzahlBegrenzung2 : {REDUND_UNREPLICABLE} REAL;
		DrehzahlBegrenzung3 : {REDUND_UNREPLICABLE} REAL;
	END_VAR
	VAR_OUTPUT
		StrombegrenzungEin : {REDUND_UNREPLICABLE} BOOL;
		DrehzahlBegrenzung : {REDUND_UNREPLICABLE} REAL;
	END_VAR
	VAR
		FreigZeitfenster1 : {REDUND_UNREPLICABLE} BOOL;
		FreigZeitfenster2 : {REDUND_UNREPLICABLE} BOOL;
		FreigZeitfenster3 : {REDUND_UNREPLICABLE} BOOL;
	END_VAR
END_FUNCTION_BLOCK

{REDUND_UNREPLICABLE} FUNCTION_BLOCK fbTrockAutomatik (*Trocknung im Automatikbetrieb*) (*$GROUP=Anwender*)
	VAR_INPUT
		Freigabe : {REDUND_UNREPLICABLE} BOOL;
		WetterIstGut : {REDUND_UNREPLICABLE} BOOL;
		LuftaufberVhd : {REDUND_UNREPLICABLE} BOOL;
		Tick : {REDUND_UNREPLICABLE} BOOL;
		LaufzeitSchlecht : {REDUND_UNREPLICABLE} UDINT;
		LaufzeitSchlechtMin : {REDUND_UNREPLICABLE} UDINT;
		PausenzeitSchlecht : {REDUND_UNREPLICABLE} UDINT;
	END_VAR
	VAR_OUTPUT
		FreigabeAutomatik : {REDUND_UNREPLICABLE} BOOL;
		Intervallbetrieb : {REDUND_UNREPLICABLE} BOOL;
	END_VAR
	VAR
		fbLaufPause : {REDUND_UNREPLICABLE} fbTrockLaufPause;
	END_VAR
END_FUNCTION_BLOCK

{REDUND_UNREPLICABLE} FUNCTION_BLOCK fbTrockStufen (*Umschaltung der Trockenstufen*) (*$GROUP=Anwender*)
	VAR_INPUT
		Freigabe : {REDUND_UNREPLICABLE} BOOL;
		FeuchteStufen : {REDUND_UNREPLICABLE} ARRAY[0..10] OF REAL;
		FeuchteStart : {REDUND_UNREPLICABLE} REAL;
		VerzStufenwechsel : {REDUND_UNREPLICABLE} UDINT;
		Bestaetigung : {REDUND_UNREPLICABLE} BOOL;
		FeuchteAktuell : {REDUND_UNREPLICABLE} REAL;
		FeuchteEnde : {REDUND_UNREPLICABLE} REAL; (*Gewünschte Feuchte bei Trocknungsende*)
		NachtrocknungFertig : {REDUND_UNREPLICABLE} BOOL;
		AktuelleRezeptNr : {REDUND_UNREPLICABLE} USINT; (*Aktuell gesetztes Rezept*)
		FreigabeAuto : {REDUND_UNREPLICABLE} BOOL; (*Freigabe im Automatikbetrieb*)
	END_VAR
	VAR_OUTPUT
		RezeptStufeIst : {REDUND_UNREPLICABLE} INT;
		MldgBestaetigungErforderl : {REDUND_UNREPLICABLE} BOOL;
		RezeptStufeBeiEnde : {REDUND_UNREPLICABLE} INT;
		MeldungFertig : {REDUND_UNREPLICABLE} BOOL; (*Meldung Trocknungsende erreicht*)
	END_VAR
	VAR
		i : {REDUND_UNREPLICABLE} INT;
		RezeptStufeSoll : {REDUND_UNREPLICABLE} INT;
		fbLascoZdxx_0 : {REDUND_UNREPLICABLE} fbLascoZdxx;
		TickStufe : {REDUND_UNREPLICABLE} BOOL;
		Stufe6_ok : {REDUND_UNREPLICABLE} BOOL;
		TON_AenderungStufeAuto : {REDUND_UNREPLICABLE} TON;
	END_VAR
END_FUNCTION_BLOCK

{REDUND_UNREPLICABLE} FUNCTION_BLOCK fbTrockVent (*Ansteuerung, Ventilatoren, Luftentfeuchter und Klappen*) (*$GROUP=Anwender*)
	VAR_INPUT
		Freigabe : {REDUND_UNREPLICABLE} BOOL;
		AnfVent1 : {REDUND_UNREPLICABLE} BOOL;
		AnfVent2 : {REDUND_UNREPLICABLE} BOOL;
		AnfLuftentf : {REDUND_UNREPLICABLE} BOOL;
		Tarifabschaltung : {REDUND_UNREPLICABLE} BOOL;
		Strombegrenzung : {REDUND_UNREPLICABLE} BOOL;
		IstDrehzahlVent1 : {REDUND_UNREPLICABLE} REAL;
		IstDrehzahlVent2 : {REDUND_UNREPLICABLE} REAL;
		DrehzahlVent1Max : {REDUND_UNREPLICABLE} REAL;
		DrehzahlVent2Max : {REDUND_UNREPLICABLE} REAL;
		DrehzahlVent1Leistung : {REDUND_UNREPLICABLE} REAL;
		DrehzahlVent2Leistung : {REDUND_UNREPLICABLE} REAL;
		DrehzahlBeiStrombegrenzung : {REDUND_UNREPLICABLE} REAL;
		AnlaufverzVent2 : {REDUND_UNREPLICABLE} UDINT;
		LaufzeitKlappen : {REDUND_UNREPLICABLE} UDINT;
		AuslaufzeitLuftentfeuchter : {REDUND_UNREPLICABLE} UDINT;
		MessdauerLuftgeschw : {REDUND_UNREPLICABLE} UDINT;
		sekTick : {REDUND_UNREPLICABLE} BOOL;
		LuftgeschwBeiMaxDrehzahl1Vent : REFERENCE TO REAL;
		LuftgeschwBeiMaxDrehzahl2Vent : REFERENCE TO REAL;
		LuftgeschwAktuell : {REDUND_UNREPLICABLE} REAL;
		KeineKlappenAmLuftentf : {REDUND_UNREPLICABLE} BOOL;
		EinschaltverzLuftentf : {REDUND_UNREPLICABLE} UDINT;
		BetriebsmldgLuftentf : {REDUND_UNREPLICABLE} BOOL; (*Betriebsmeldung von Luftentfeuchter*)
	END_VAR
	VAR_OUTPUT
		curStep : {REDUND_UNREPLICABLE} enumStepTrockVent;
		FreigabeKlappen : {REDUND_UNREPLICABLE} BOOL;
		FreigabeLuftentf : {REDUND_UNREPLICABLE} BOOL;
		FreigabeVent1 : {REDUND_UNREPLICABLE} BOOL;
		FreigabeVent2 : {REDUND_UNREPLICABLE} BOOL;
		TON_AnlaufverzVent2 : {REDUND_UNREPLICABLE} TON;
		TON_LaufzeitKlappen : {REDUND_UNREPLICABLE} TON;
		SollDrehzVent1 : {REDUND_UNREPLICABLE} REAL;
		SollDrehzVent2 : {REDUND_UNREPLICABLE} REAL;
		TON_AuslaufzeitLuftentf : {REDUND_UNREPLICABLE} TON;
		TON_Messung : {REDUND_UNREPLICABLE} TON;
		MessungAktiv : {REDUND_UNREPLICABLE} BOOL;
		TON_LuftentfVorbereitung : {REDUND_UNREPLICABLE} TON;
	END_VAR
	VAR
		nextStep : {REDUND_UNREPLICABLE} enumStepTrockVent;
		stateEntry : {REDUND_UNREPLICABLE} BOOL;
		Mittelwertbildung : {REDUND_UNREPLICABLE} LCRMovAvgFlt;
	END_VAR
END_FUNCTION_BLOCK

{REDUND_UNREPLICABLE} FUNCTION_BLOCK fbTrockVariante (*Auswertung der Anlagenkonfiguration mit Ausgabe einer Nummer und eines Textes*) (*$GROUP=Anwender*)
	VAR_INPUT
		Freigabe : {REDUND_UNREPLICABLE} BOOL;
		Ventilator1 : {REDUND_UNREPLICABLE} BOOL;
		Ventilator2 : {REDUND_UNREPLICABLE} BOOL;
		Luftentfeuchter : {REDUND_UNREPLICABLE} BOOL;
		Warmluftofen : {REDUND_UNREPLICABLE} BOOL;
		BetriebsmldgWarmluftofen : {REDUND_UNREPLICABLE} BOOL;
		BetriebsmldgScheitholzofen : {REDUND_UNREPLICABLE} BOOL;
		Brandschutzklappe : {REDUND_UNREPLICABLE} BOOL;
		Umschaltklappe : {REDUND_UNREPLICABLE} BOOL;
	END_VAR
	VAR_OUTPUT
		VarianteNr : {REDUND_UNREPLICABLE} USINT;
		VarianteName : {REDUND_UNREPLICABLE} STRING[200];
	END_VAR
END_FUNCTION_BLOCK
```

#### fbTrockZeitprogramm.st - Generierung von Start- und Stoppsignalen aus Zeitprogramm
```iecst
(********************************************************************
 * COPYRIGHT -- LASCO Heu- und Forsttechnik GmbH
 ********************************************************************
 * Library: LascoTrock
 * Datei: fbTrockZeitprogramm.st
 * Autor: Rudolf Lachner
 * Erstellt: 10. März 2014
 ********************************************************************
 * Implementierung der Library LascoTrock
 ********************************************************************)

(* Generierung von Start- und Stoppsignalen aus Zeitprogramm *)
FUNCTION_BLOCK fbTrockZeitprogramm

	IF (Freigabe = TRUE) THEN

		//Zeitfenster 1 ****************************************************************************************************************************
		FreigZeitfenster1	:= FALSE;
		IF (StartZeit1 > StoppZeit1) THEN
			IF (AktZeit >= StartZeit1) OR (AktZeit < StoppZeit1) THEN
				FreigZeitfenster1 	:= TRUE;
			END_IF
		ELSE
			IF (AktZeit >= StartZeit1) AND (AktZeit < StoppZeit1) THEN
				FreigZeitfenster1	:= TRUE;
			END_IF
		END_IF

		//Zeitfenster 2 ****************************************************************************************************************************
		FreigZeitfenster2	:= FALSE;
		IF (StartZeit2 > StoppZeit2) THEN
			IF (AktZeit >= StartZeit2) OR (AktZeit < StoppZeit2) THEN
				FreigZeitfenster2 	:= TRUE;
			END_IF
		ELSE
			IF (AktZeit >= StartZeit2) AND (AktZeit < StoppZeit2) THEN
				FreigZeitfenster2	:= TRUE;
			END_IF
		END_IF

		//Zeitfenster 3 ****************************************************************************************************************************
		FreigZeitfenster3	:= FALSE;
		IF (StartZeit3 > StoppZeit3) THEN
			IF (AktZeit >= StartZeit3) OR (AktZeit < StoppZeit3) THEN
				FreigZeitfenster3 	:= TRUE;
			END_IF
		ELSE
			IF (AktZeit >= StartZeit3) AND (AktZeit < StoppZeit3) THEN
				FreigZeitfenster3	:= TRUE;
			END_IF
		END_IF

		//Zeitfenster 4 ****************************************************************************************************************************
		FreigZeitfenster4	:= FALSE;
		IF (StartZeit4 > StoppZeit4) THEN
			IF (AktZeit >= StartZeit4) OR (AktZeit < StoppZeit4) THEN
				FreigZeitfenster4 	:= TRUE;
			END_IF
		ELSE
			IF (AktZeit >= StartZeit4) AND (AktZeit < StoppZeit4) THEN
				FreigZeitfenster4	:= TRUE;
			END_IF
		END_IF

		//Zeitfenster 5 ****************************************************************************************************************************
		FreigZeitfenster5	:= FALSE;
		IF (StartZeit5 > StoppZeit5) THEN
			IF (AktZeit >= StartZeit5) OR (AktZeit < StoppZeit5) THEN
				FreigZeitfenster5 	:= TRUE;
			END_IF
		ELSE
			IF (AktZeit >= StartZeit5) AND (AktZeit < StoppZeit5) THEN
				FreigZeitfenster5	:= TRUE;
			END_IF
		END_IF

		FreigabeZeitprogramm	:= FreigZeitfenster1 OR FreigZeitfenster2 OR FreigZeitfenster3 OR FreigZeitfenster4 OR FreigZeitfenster5;

	ELSE

		FreigZeitfenster1		:= FALSE;
		FreigZeitfenster2		:= FALSE;
		FreigZeitfenster3		:= FALSE;
		FreigZeitfenster4		:= FALSE;
		FreigZeitfenster5		:= FALSE;
		FreigabeZeitprogramm	:= FALSE;

	END_IF

END_FUNCTION_BLOCK
```

#### fbTrockLaufPause.st - Lauf- und Pausenprogramm
```iecst
(********************************************************************
 * COPYRIGHT -- LASCO Heu- und Forsttechnik GmbH
 ********************************************************************
 * Library: LascoTrock
 * Datei: fbTrockLaufPause.st
 * Autor: Rudolf Lachner
 * Erstellt: 18. März 2014
 ********************************************************************
 * Implementierung der Library LascoTrock
 ********************************************************************)

(* Lauf- und Pausenprogramm *)
FUNCTION_BLOCK fbTrockLaufPause

	//Schrittschaltwerk Pulsgenerator
	//===============================

	currStep	:= nextStep;

	CASE currStep OF

		//*******************************************************************************************************************************************************************************
		0://WARTEN

			//*** state during ***
			FreigabeLpPrg	:= FALSE;

			CounterLauf		:= 0;
			CounterPause	:= 0;
			RestzeitPause	:= 0;
			RestzeitLauf	:= 0;

			//*** state exit ***
			IF (Freigabe) AND (ZeitLauf <> 0) AND (ZeitLauf >= ZeitLaufMin) AND NOT (Reset) THEN
				nextStep	:= 2;
			ELSE
				nextStep	:= currStep;
			END_IF

		//***********************************************************************************************************************************************************************************
		1://PAUSE

			//*** state during ***
			FreigabeLpPrg	:= FALSE;

			IF (EDGEPOS(Tick)) THEN
				CounterPause	:= CounterPause + 1;
			END_IF

			RestzeitPause	:= ZeitPause - CounterPause;
			RestzeitLauf	:= 0;

			//*** state exit ***
			IF (NOT Freigabe) OR (ZeitLauf = 0) OR (ZeitLauf < ZeitLaufMin) OR (Reset) THEN
				nextStep	:= 0;
			ELSIF (CounterPause >= ZeitPause) THEN
				CounterPause	:= 0;
				nextStep		:= 2;
			END_IF

		//************************************************************************************************************************************************************************************************
		2://LAUF

			//*** state during ***
			FreigabeLpPrg	:= TRUE;

			IF (EDGEPOS(Tick)) THEN
				CounterLauf		:= CounterLauf + 1;
			END_IF

			RestzeitPause	:= 0;
			RestzeitLauf	:= ZeitLauf - CounterLauf;

			//*** state exit ***
			IF (NOT Freigabe) OR (ZeitLauf < ZeitLaufMin) OR (Reset) THEN
				nextStep	:= 0;
			ELSIF (CounterLauf >= ZeitLauf) THEN
				CounterLauf	:= 0;
				nextStep	:= 1;
			END_IF

	END_CASE

END_FUNCTION_BLOCK
```

#### fbTrockNachtrock.st - Funktionsbaustein Nachtrocknung
```iecst
(********************************************************************
 * COPYRIGHT -- LASCO Heu- und Forsttechnik GmbH
 ********************************************************************
 * Library: LascoTrock
 * Datei: fbTrockNachtrock.st
 * Autor: Rudolf Lachner
 * Erstellt: 18. März 2014
 ********************************************************************
 * Implementierung der Library LascoTrock
 ********************************************************************)

(* Funktionsbaustein Nachtrocknung *)
FUNCTION_BLOCK fbTrockNachtrock

	IF (Freigabe = TRUE) THEN

		//Zeitfenster 1 ****************************************************************************************************************************
		FreigZeitfenster1	:= FALSE;
		IF (StartZeit1 > StoppZeit1) THEN
			IF (AktZeit >= StartZeit1) OR (AktZeit < StoppZeit1) THEN
				FreigZeitfenster1 	:= TRUE;
			END_IF
		ELSE
			IF (AktZeit >= StartZeit1) AND (AktZeit < StoppZeit1) THEN
				FreigZeitfenster1	:= TRUE;
			END_IF
		END_IF

		//Zeitfenster 2 ****************************************************************************************************************************
		FreigZeitfenster2	:= FALSE;
		IF (StartZeit2 > StoppZeit2) THEN
			IF (AktZeit >= StartZeit2) OR (AktZeit < StoppZeit2) THEN
				FreigZeitfenster2 	:= TRUE;
			END_IF
		ELSE
			IF (AktZeit >= StartZeit2) AND (AktZeit < StoppZeit2) THEN
				FreigZeitfenster2	:= TRUE;
			END_IF
		END_IF

		//Zeitfenster 3 ****************************************************************************************************************************
		FreigZeitfenster3	:= FALSE;
		IF (StartZeit3 > StoppZeit3) THEN
			IF (AktZeit >= StartZeit3) OR (AktZeit < StoppZeit3) THEN
				FreigZeitfenster3 	:= TRUE;
			END_IF
		ELSE
			IF (AktZeit >= StartZeit3) AND (AktZeit < StoppZeit3) THEN
				FreigZeitfenster3	:= TRUE;
			END_IF
		END_IF

		//Dauer Nachtrocknung mitzählen
		IF (TagTick) THEN
			TageNachtrocknungAktiv	:= TageNachtrocknungAktiv + 1;
			ZyklusTageIst			:= ZyklusTageIst + 1;
			AktTagFreigabe			:= FALSE;
		END_IF

		IF StdTick THEN
			StdNachtrocknung		:= StdNachtrocknung + 1;
		END_IF

		//Wenn Zyklus Nachtrocknung erreicht -> Freigabe
		IF (ZyklusTageIst >= ZyklusTageSoll) THEN
			AktTagFreigabe			:= TRUE;
			ZyklusTageIst			:= 0;
		END_IF

		//Meldung Nachtrocknung Fertig
		IF (TageNachtrocknungAktiv >= DauerNachtrocknungTage) THEN
			NachtrocknungFertig		:= TRUE;
		ELSE
			NachtrocknungFertig		:= FALSE;
		END_IF

		FreigabeNachtrocknung	:= (FreigZeitfenster1 OR FreigZeitfenster2 OR FreigZeitfenster3) AND ((AktTagFreigabe) OR (TageNachtrocknungAktiv = 0)) ;

	ELSE

		FreigZeitfenster1		:= FALSE;
		FreigZeitfenster2		:= FALSE;
		FreigZeitfenster3		:= FALSE;
		FreigabeNachtrocknung	:= FALSE;
		AktTagFreigabe			:= FALSE;
		NachtrocknungFertig		:= FALSE;
		ZyklusTageIst			:= 0;
		TageNachtrocknungAktiv	:= 0;
		StdNachtrocknung		:= 0;

	END_IF

END_FUNCTION_BLOCK
```

#### fbTrockTarifabsch.st - Funktionsbaustein Tarifabschaltung
```iecst
(* Funktionsbaustein Tarifabschaltung *)
FUNCTION_BLOCK fbTrockTarifabsch

	IF (Freigabe = TRUE) THEN

		//Zeitfenster 1 ****************************************************************************************************************************

		StartZeit1	:= (StartStd1 * 100) + StartMin1;
		StoppZeit1	:= (StoppStd1 * 100) + StoppMin1;

		//Vorlaufzeit Luftaufbereitung berechnen
		loc_StdVorlaufzeitREAL 	:= VorlaufzeitLuftaufbMin / 60;
		loc_StdVorlaufzeit		:= TRUNC(loc_StdVorlaufzeitREAL);

		loc_MinVorlaufzeit	:= VorlaufzeitLuftaufbMin - (loc_StdVorlaufzeit * 60);

		loc_ZwischenergStartStd	:= StartStd1 - loc_StdVorlaufzeit;
		IF (loc_ZwischenergStartStd < 0) THEN
			loc_StartStdLuftaufb	:= 24 + loc_ZwischenergStartStd;
		ELSE
			loc_StartStdLuftaufb	:= loc_ZwischenergStartStd;
		END_IF

		loc_ZwischenergStartMin := StartMin1 - loc_MinVorlaufzeit;
		IF loc_ZwischenergStartMin < 0 THEN
			loc_StartMinLuftaufb	:= 60 + loc_ZwischenergStartMin;
			loc_StartStdLuftaufb	:= loc_StartStdLuftaufb - 1;
			IF (loc_StartStdLuftaufb < 0) THEN
				loc_StartStdLuftaufb	:= 24 + loc_StartStdLuftaufb;
			END_IF
		ELSE
			loc_StartMinLuftaufb	:= loc_ZwischenergStartMin;
		END_IF

		StartZeitLuftaufb1	:= (loc_StartStdLuftaufb * 100) + loc_StartMinLuftaufb;

		//Freigabe Zeitfenster 1
		FreigZeitfenster1	:= FALSE;
		IF (StartZeit1 > StoppZeit1) THEN
			IF (AktZeit >= StartZeit1) OR (AktZeit < StoppZeit1) THEN
				FreigZeitfenster1 	:= TRUE;
			END_IF
		ELSE
			IF (AktZeit >= StartZeit1) AND (AktZeit < StoppZeit1) THEN
				FreigZeitfenster1	:= TRUE;
			END_IF
		END_IF

		//Freigabe Zeitfenster Luftaufbereitung 1
		FreigabeZeitfensterLuftaufb1	:= FALSE;
		IF (StartZeit1 <> 0) AND (StoppZeit1 <> 0) THEN
			IF (StartZeitLuftaufb1 > StoppZeit1) THEN
				IF (AktZeit >= StartZeitLuftaufb1) OR (AktZeit < StoppZeit1) THEN
					FreigabeZeitfensterLuftaufb1	:= TRUE;
				END_IF
			ELSE
				IF (AktZeit >= StartZeitLuftaufb1) AND (AktZeit < StoppZeit1) THEN
					FreigabeZeitfensterLuftaufb1	:= TRUE;
				END_IF
			END_IF
		END_IF

		//Zeitfenster 2 ****************************************************************************************************************************

		StartZeit2	:= (StartStd2 * 100) + StartMin2;
		StoppZeit2	:= (StoppStd2 * 100) + StoppMin2;

		//Vorlaufzeit Luftaufbereitung berechnen
		loc_StdVorlaufzeitREAL 	:= VorlaufzeitLuftaufbMin / 60;
		loc_StdVorlaufzeit		:= TRUNC(loc_StdVorlaufzeitREAL);

		loc_MinVorlaufzeit	:= VorlaufzeitLuftaufbMin - (loc_StdVorlaufzeit * 60);

		loc_ZwischenergStartStd	:= StartStd2 - loc_StdVorlaufzeit;
		IF (loc_ZwischenergStartStd < 0) THEN
			loc_StartStdLuftaufb	:= 24 + loc_ZwischenergStartStd;
		ELSE
			loc_StartStdLuftaufb	:= loc_ZwischenergStartStd;
		END_IF

		loc_ZwischenergStartMin := StartMin2 - loc_MinVorlaufzeit;
		IF loc_ZwischenergStartMin < 0 THEN
			loc_StartMinLuftaufb	:= 60 + loc_ZwischenergStartMin;
			loc_StartStdLuftaufb	:= loc_StartStdLuftaufb - 1;
			IF (loc_StartStdLuftaufb < 0) THEN
				loc_StartStdLuftaufb	:= 24 + loc_StartStdLuftaufb;
			END_IF
		ELSE
			loc_StartMinLuftaufb	:= loc_ZwischenergStartMin;
		END_IF

		StartZeitLuftaufb2	:= (loc_StartStdLuftaufb * 100) + loc_StartMinLuftaufb;

		//Freigabe Zeitfenster 2
		FreigZeitfenster2	:= FALSE;
		IF (StartZeit2 > StoppZeit2) THEN
			IF (AktZeit >= StartZeit2) OR (AktZeit < StoppZeit2) THEN
				FreigZeitfenster2 	:= TRUE;
			END_IF
		ELSE
			IF (AktZeit >= StartZeit2) AND (AktZeit < StoppZeit2) THEN
				FreigZeitfenster2	:= TRUE;
			END_IF
		END_IF

		//Freigabe Zeitfenster Luftaufbereitung 2
		FreigabeZeitfensterLuftaufb2	:= FALSE;
		IF (StartZeit2 <> 0) AND (StoppZeit2 <> 0) THEN
			IF (StartZeitLuftaufb2 > StoppZeit2) THEN
				IF (AktZeit >= StartZeitLuftaufb2) OR (AktZeit < StoppZeit2) THEN
					FreigabeZeitfensterLuftaufb2	:= TRUE;
				END_IF
			ELSE
				IF (AktZeit >= StartZeitLuftaufb2) AND (AktZeit < StoppZeit2) THEN
					FreigabeZeitfensterLuftaufb2	:= TRUE;
				END_IF
			END_IF
		END_IF

		//Zeitfenster 3 ****************************************************************************************************************************

		StartZeit3	:= (StartStd3 * 100) + StartMin3;
		StoppZeit3	:= (StoppStd3 * 100) + StoppMin3;

		//Vorlaufzeit Luftaufbereitung berechnen
		loc_StdVorlaufzeitREAL 	:= VorlaufzeitLuftaufbMin / 60;
		loc_StdVorlaufzeit		:= TRUNC(loc_StdVorlaufzeitREAL);

		loc_MinVorlaufzeit	:= VorlaufzeitLuftaufbMin - (loc_StdVorlaufzeit * 60);

		loc_ZwischenergStartStd	:= StartStd3 - loc_StdVorlaufzeit;
		IF (loc_ZwischenergStartStd < 0) THEN
			loc_StartStdLuftaufb	:= 24 + loc_ZwischenergStartStd;
		ELSE
			loc_StartStdLuftaufb	:= loc_ZwischenergStartStd;
		END_IF

		loc_ZwischenergStartMin := StartMin3 - loc_MinVorlaufzeit;
		IF loc_ZwischenergStartMin < 0 THEN
			loc_StartMinLuftaufb	:= 60 + loc_ZwischenergStartMin;
			loc_StartStdLuftaufb	:= loc_StartStdLuftaufb - 1;
			IF (loc_StartStdLuftaufb < 0) THEN
				loc_StartStdLuftaufb	:= 24 + loc_StartStdLuftaufb;
			END_IF
		ELSE
			loc_StartMinLuftaufb	:= loc_ZwischenergStartMin;
		END_IF

		StartZeitLuftaufb3	:= (loc_StartStdLuftaufb * 100) + loc_StartMinLuftaufb;

		//Freigabe Zeitfenster 3
		FreigZeitfenster3	:= FALSE;
		IF (StartZeit3 > StoppZeit3) THEN
			IF (AktZeit >= StartZeit3) OR (AktZeit < StoppZeit3) THEN
				FreigZeitfenster3 	:= TRUE;
			END_IF
		ELSE
			IF (AktZeit >= StartZeit3) AND (AktZeit < StoppZeit3) THEN
				FreigZeitfenster3	:= TRUE;
			END_IF
		END_IF

		//Freigabe Zeitfenster Luftaufbereitung 3
		FreigabeZeitfensterLuftaufb3	:= FALSE;
		IF (StartZeit3 <> 0) AND (StoppZeit3 <> 0) THEN
			IF (StartZeitLuftaufb3 > StoppZeit3) THEN
				IF (AktZeit >= StartZeitLuftaufb3) OR (AktZeit < StoppZeit3) THEN
					FreigabeZeitfensterLuftaufb3	:= TRUE;
				END_IF
			ELSE
				IF (AktZeit >= StartZeitLuftaufb3) AND (AktZeit < StoppZeit3) THEN
					FreigabeZeitfensterLuftaufb3	:= TRUE;
				END_IF
			END_IF
		END_IF

		TarifabschaltungEin			:= FreigZeitfenster1 OR FreigZeitfenster2 OR FreigZeitfenster3;
		TarifabschaltungLuftaufbEin	:= FreigabeZeitfensterLuftaufb1 OR FreigabeZeitfensterLuftaufb2 OR FreigabeZeitfensterLuftaufb3;

	ELSE

		FreigZeitfenster1				:= FALSE;
		FreigZeitfenster2				:= FALSE;
		FreigZeitfenster3				:= FALSE;
		FreigabeZeitfensterLuftaufb1	:= FALSE;
		FreigabeZeitfensterLuftaufb2	:= FALSE;
		FreigabeZeitfensterLuftaufb3	:= FALSE;
		TarifabschaltungEin				:= FALSE;
		TarifabschaltungLuftaufbEin		:= FALSE;
		loc_MinVorlaufzeit				:= 0;
		loc_StartMinLuftaufb			:= 0;
		loc_StartStdLuftaufb			:= 0;
		loc_StdVorlaufzeit				:= 0;
		loc_StdVorlaufzeitREAL			:= 0;
		loc_ZwischenergStartMin			:= 0;
		loc_ZwischenergStartStd			:= 0;

	END_IF

END_FUNCTION_BLOCK
```

#### fbTrockStrombegr.st - Strombegrenzung in bestimmten Zeitfenstern
```iecst
(********************************************************************
 * COPYRIGHT -- LASCO Heu- und Forsttechnik GmbH
 ********************************************************************
 * Library: LascoTrock
 * Datei: fbTrockStrombegr.st
 * Autor: Rudolf Lachner
 * Erstellt: 18. März 2014
 ********************************************************************
 * Implementierung der Library LascoTrock
 ********************************************************************)

(* Strombegrenzung in bestimmten Zeitfenstern *)
FUNCTION_BLOCK fbTrockStrombegr

	IF (Freigabe = TRUE) THEN

		//Zeitfenster 1 ****************************************************************************************************************************
		FreigZeitfenster1	:= FALSE;
		IF (StartZeit1 > StoppZeit1) THEN
			IF (AktZeit >= StartZeit1) OR (AktZeit < StoppZeit1) THEN
				FreigZeitfenster1 	:= TRUE;
			END_IF
		ELSE
			IF (AktZeit >= StartZeit1) AND (AktZeit < StoppZeit1) THEN
				FreigZeitfenster1	:= TRUE;
			END_IF
		END_IF

		//Zeitfenster 2 ****************************************************************************************************************************
		FreigZeitfenster2	:= FALSE;
		IF (StartZeit2 > StoppZeit2) THEN
			IF (AktZeit >= StartZeit2) OR (AktZeit < StoppZeit2) THEN
				FreigZeitfenster2 	:= TRUE;
			END_IF
		ELSE
			IF (AktZeit >= StartZeit2) AND (AktZeit < StoppZeit2) THEN
				FreigZeitfenster2	:= TRUE;
			END_IF
		END_IF

		//Zeitfenster 3 ****************************************************************************************************************************
		FreigZeitfenster3	:= FALSE;
		IF (StartZeit3 > StoppZeit3) THEN
			IF (AktZeit >= StartZeit3) OR (AktZeit < StoppZeit3) THEN
				FreigZeitfenster3 	:= TRUE;
			END_IF
		ELSE
			IF (AktZeit >= StartZeit3) AND (AktZeit < StoppZeit3) THEN
				FreigZeitfenster3	:= TRUE;
			END_IF
		END_IF

		//Drehzahlbegrenzungen 1 - 3
		//**************************
		IF (FreigZeitfenster1) THEN
			DrehzahlBegrenzung	:= DrehzahlBegrenzung1;
		ELSIF (FreigZeitfenster2) THEN
			DrehzahlBegrenzung	:= DrehzahlBegrenzung2;
		ELSIF (FreigZeitfenster3) THEN
			DrehzahlBegrenzung	:= DrehzahlBegrenzung3;
		ELSE
			DrehzahlBegrenzung	:= 0.0;
		END_IF

		StrombegrenzungEin		:= FreigZeitfenster1 OR FreigZeitfenster2 OR FreigZeitfenster3;

	ELSE

		FreigZeitfenster1		:= FALSE;
		FreigZeitfenster2		:= FALSE;
		FreigZeitfenster3		:= FALSE;
		StrombegrenzungEin		:= FALSE;
		DrehzahlBegrenzung		:= 0.0;

	END_IF

END_FUNCTION_BLOCK
```

#### fbTrockAutomatik.st - Trocknung im Automatikbetrieb
```iecst
(********************************************************************
 * COPYRIGHT -- LASCO Heu- und Forsttechnik GmbH
 ********************************************************************
 * Library: LascoTrock
 * Datei: fbTrockAutomatik.st
 * Autor: Rudolf Lachner
 * Erstellt: 18. März 2014
 ********************************************************************
 * Implementierung der Library LascoTrock
 ********************************************************************)

(* Trocknung im Automatikbetrieb *)
FUNCTION_BLOCK fbTrockAutomatik

	IF (Freigabe = TRUE) THEN

		IF (WetterIstGut OR LuftaufberVhd) THEN
			Intervallbetrieb		:= FALSE;
			FreigabeAutomatik		:= TRUE;
			fbLaufPause.Freigabe	:= FALSE;
			fbLaufPause.Reset		:= TRUE;
		ELSE
			Intervallbetrieb		:= TRUE;
			fbLaufPause.Freigabe	:= TRUE;
			fbLaufPause.Tick		:= Tick;
			fbLaufPause.Reset		:= FALSE;
			fbLaufPause.ZeitLauf	:= LaufzeitSchlecht;
			fbLaufPause.ZeitLaufMin	:= LaufzeitSchlechtMin;
			fbLaufPause.ZeitPause	:= PausenzeitSchlecht;
			fbLaufPause();
			FreigabeAutomatik		:= fbLaufPause.FreigabeLpPrg;
		END_IF
	ELSE
		Intervallbetrieb		:= FALSE;
		FreigabeAutomatik		:= FALSE;
		fbLaufPause.Freigabe	:= FALSE;
		fbLaufPause.Reset		:= TRUE;
		fbLaufPause();
	END_IF

END_FUNCTION_BLOCK
```

#### fbTrockStufen.st - Umschaltung der Trockenstufen
```iecst
(********************************************************************
 * COPYRIGHT -- LASCO Heu- und Forsttechnik GmbH
 ********************************************************************
 * Library: LascoTrock
 * Datei: fbTrockStufen.st
 * Autor: Rudolf Lachner
 * Erstellt: 19. März 2014
 ********************************************************************
 * Implementierung der Library LascoTrock
 ********************************************************************)

(* Umschaltung der Trockenstufen *)
FUNCTION_BLOCK fbTrockStufen

	//Freigabe, Automatik ***************************************************************************************************************
	IF (Freigabe = TRUE) AND (FreigabeAuto = TRUE) AND (AktuelleRezeptNr <> 0) THEN

		//Bei Trocknungsstart auf Stufe Startfeuchte setzen
		//*************************************************
		IF (FeuchteStart > 0) AND (RezeptStufeIst = 0) THEN
			FOR i := 1 TO 6 DO
				IF (FeuchteStart <= FeuchteStufen[i]) THEN
					RezeptStufeSoll	:= i;
					RezeptStufeIst	:= i;
				END_IF
				IF (FeuchteStart > FeuchteStufen[1]) THEN
					RezeptStufeIst		:= 1;
					RezeptStufeSoll		:= 1;
				END_IF
			END_FOR
		END_IF

		//Passende Stufe ermitteln
		FOR i := 1 TO 6 DO
			IF (FeuchteAktuell <= FeuchteStufen[i]) THEN
				RezeptStufeSoll	:= i;
			END_IF
		END_FOR
		IF (FeuchteAktuell > FeuchteStufen[1]) THEN
			RezeptStufeSoll		:= 1;
		END_IF

		//Tick bei Änderung der Sollstufe
		fbLascoZdxx_0(IN 	:= RezeptStufeSoll);
		TickStufe			:= fbLascoZdxx_0.Q;

		//Zeitverzögerung Übernahme Änderung Stufe (Stufe 1 bis 5)
		IF (RezeptStufeSoll <= 5) THEN

			Stufe6_ok	:= FALSE;

			TON_AenderungStufeAuto.IN	:= (RezeptStufeSoll <> RezeptStufeIst) AND NOT TickStufe;
			TON_AenderungStufeAuto.PT	:= UDINT_TO_TIME(VerzStufenwechsel);
			TON_AenderungStufeAuto();

			IF (TON_AenderungStufeAuto.Q) THEN
				RezeptStufeIst := RezeptStufeSoll;
			END_IF
		END_IF

		//Bestätigung für das Umschalten von Stufe 5 auf 6 notwendig
		IF (RezeptStufeSoll = 6) AND NOT (Stufe6_ok) THEN
			MldgBestaetigungErforderl	:= TRUE;
			IF (Bestaetigung) THEN
				RezeptStufeIst := RezeptStufeSoll;
				Stufe6_ok		:= TRUE;
			END_IF
		ELSE
			MldgBestaetigungErforderl	:= FALSE;
		END_IF

		//Stufe bei Trocknungsende ermitteln
		FOR i := 1 TO 6 DO
			IF (FeuchteEnde <= FeuchteStufen[i]) AND (FeuchteEnde > 0) THEN
				RezeptStufeBeiEnde	:= i;
			ELSIF (FeuchteEnde > 0) AND (FeuchteStufen[i] <= FeuchteEnde) AND NOT (FeuchteEnde > FeuchteStufen[i]) THEN
				RezeptStufeBeiEnde	:= i;
			END_IF
		END_FOR

		//Meldung Trocknung Fertig ausgeben
		//*********************************

		MeldungFertig	:= FALSE;

		IF (RezeptStufeBeiEnde < 6) THEN
			IF (RezeptStufeIst >= RezeptStufeBeiEnde) THEN
				MeldungFertig	:= TRUE;
			END_IF
		ELSIF (RezeptStufeBeiEnde >= 6) THEN
			IF (NachtrocknungFertig) THEN
				MeldungFertig	:= TRUE;
			END_IF
		END_IF

	//Freigabe ********************************************************************************************************************************
	ELSIF (Freigabe = TRUE) AND (AktuelleRezeptNr <> 0) THEN

		//Bei Trocknungsstart auf Stufe Startfeuchte setzen
		//*************************************************
		IF (FeuchteStart > 0) AND (RezeptStufeIst = 0) THEN
			FOR i := 1 TO 6 DO
				IF (FeuchteStart <= FeuchteStufen[i]) THEN
					RezeptStufeSoll	:= i;
					RezeptStufeIst	:= i;
				END_IF
				IF (FeuchteStart > FeuchteStufen[1]) THEN
					RezeptStufeIst		:= 1;
					RezeptStufeSoll		:= 1;
				END_IF
			END_FOR
		END_IF

		//Passende Stufe ermitteln
		FOR i := 1 TO 6 DO
			IF (FeuchteAktuell <= FeuchteStufen[i]) THEN
				RezeptStufeSoll	:= i;
			END_IF
		END_FOR
		IF (FeuchteAktuell > FeuchteStufen[1]) THEN
			RezeptStufeSoll		:= 1;
		END_IF

		//Tick bei Änderung der Sollstufe
		fbLascoZdxx_0(IN 	:= RezeptStufeSoll);
		TickStufe			:= fbLascoZdxx_0.Q;

		//Zeitverzögerung Übernahme Änderung Stufe (Stufe 1 bis 6) -> keine Nachtrocknung
		IF (RezeptStufeSoll <= 6) THEN
			Stufe6_ok	:= FALSE;

			TON_AenderungStufeAuto.IN	:= (RezeptStufeSoll <> RezeptStufeIst) AND NOT TickStufe;
			TON_AenderungStufeAuto.PT	:= UDINT_TO_TIME(VerzStufenwechsel);
			TON_AenderungStufeAuto();

			IF (TON_AenderungStufeAuto.Q) THEN
				RezeptStufeIst := RezeptStufeSoll;
			END_IF
		END_IF

		//Stufe bei Trocknungsende ermitteln
		FOR i := 1 TO 6 DO
			IF (FeuchteEnde <= FeuchteStufen[i]) AND (FeuchteEnde > 0) THEN
				RezeptStufeBeiEnde	:= i;
			ELSIF (FeuchteEnde > 0) AND (FeuchteStufen[i] <= FeuchteEnde) AND NOT (FeuchteEnde > FeuchteStufen[i]) THEN
				RezeptStufeBeiEnde	:= i;
			END_IF
		END_FOR

		//Meldung Trocknung Fertig ausgeben
		//*********************************
		MeldungFertig	:= FALSE;
		IF (RezeptStufeIst >= RezeptStufeBeiEnde) THEN
			MeldungFertig	:= TRUE;
		END_IF

		MldgBestaetigungErforderl	:= FALSE;

	ELSE

		MeldungFertig				:= FALSE;
		MldgBestaetigungErforderl	:= FALSE;
		RezeptStufeIst				:= 0;
		RezeptStufeBeiEnde			:= 0;
		RezeptStufeSoll				:= 0;

	END_IF

END_FUNCTION_BLOCK
```

#### fbTrockVent.st - Ansteuerung, Ventilatoren, Luftentfeuchter und Klappen
```iecst
(********************************************************************
 * COPYRIGHT -- LASCO Heu- und Forsttechnik GmbH
 ********************************************************************
 * Library: LascoTrock
 * Datei: fbTrockVent.st
 * Autor: Rudolf Lachner
 * Erstellt: 2. April 2014
 ********************************************************************
 * Implementierung der Library LascoTrock
 ********************************************************************)

(* Ansteuerung, Ventilatoren, Luftentfeuchter und Klappen *)
FUNCTION_BLOCK fbTrockVent

	IF (Freigabe = TRUE) THEN

		curStep	:= nextStep;

		CASE curStep OF

			//******************************************************************************************************************************************************************************************************************
			WARTEN_FBTROCK:

				//*** state entry ***
				IF (stateEntry) THEN
					stateEntry := FALSE;
					FreigabeKlappen		:= FALSE;
					FreigabeLuftentf	:= FALSE;
					FreigabeVent1		:= FALSE;
					FreigabeVent2		:= FALSE;
					SollDrehzVent1		:= 30.0;
					SollDrehzVent2		:= 30.0;
				END_IF

				//*** state during ***
				//Warten auf Freigabe ...

				//*** state exit ***
				IF (Tarifabschaltung) THEN
					stateEntry	:= TRUE;
					nextStep	:= TARIFABSCHALTUNG_FBTROCK;
				ELSIF ((AnfVent1 OR AnfVent2) AND NOT AnfLuftentf) THEN
					stateEntry	:= TRUE;
					nextStep	:= KLAPPEN_ZU_FBTROCK;
				ELSIF ((AnfVent1 OR AnfVent2) AND AnfLuftentf) THEN
					stateEntry	:= TRUE;
					nextStep	:= KLAPPEN_AUF_FBTROCK;
				ELSE
					nextStep	:= curStep;
				END_IF

			//******************************************************************************************************************************************************************************************************************
			VENT_EIN_FBTROCK:

				//*** state entry ***
				IF (stateEntry) THEN
					stateEntry := FALSE;
				END_IF

				//*** state during ***
				TON_AnlaufverzVent2.IN	:= FreigabeVent1;
				TON_AnlaufverzVent2.PT	:= UDINT_TO_TIME(AnlaufverzVent2);

				FreigabeVent1			:= TRUE;
				FreigabeVent2			:= AnfVent2 AND (TON_AnlaufverzVent2.Q);

				IF (Strombegrenzung AND (DrehzahlVent1Leistung >= DrehzahlBeiStrombegrenzung)) THEN
					SollDrehzVent1			:= DrehzahlBeiStrombegrenzung;
					SollDrehzVent2			:= DrehzahlBeiStrombegrenzung;
				ELSE
					SollDrehzVent1			:= DrehzahlVent1Leistung;
					SollDrehzVent2			:= DrehzahlVent2Leistung;
				END_IF

				//*** state exit ***
				IF (Tarifabschaltung) THEN
					stateEntry				:= TRUE;
					nextStep				:= TARIFABSCHALTUNG_FBTROCK;
					TON_AnlaufverzVent2.IN	:= FALSE;
				ELSIF (NOT AnfVent1 AND NOT AnfVent2) THEN
					stateEntry				:= TRUE;
					nextStep				:= VENT_AUS_FBTROCK;
					TON_AnlaufverzVent2.IN	:= FALSE;
				ELSIF (AnfLuftentf AND NOT FreigabeLuftentf) THEN
					stateEntry				:= TRUE;
					nextStep				:= KLAPPEN_AUF_FBTROCK;
					TON_AnlaufverzVent2.IN	:= FreigabeVent1;
				ELSIF (FreigabeLuftentf AND NOT AnfLuftentf) THEN
					stateEntry				:= TRUE;
					nextStep				:= LA_AUS_VORBEREITUNG_FBTROCK;
				ELSE
					nextStep				:= curStep;
				END_IF

			//******************************************************************************************************************************************************************************************************************
			VENT_AUS_FBTROCK:

				//*** state entry ***
				IF (stateEntry) THEN
					stateEntry 			:= FALSE;
					FreigabeLuftentf	:= FALSE;
				END_IF

				// *** State during	***
				SollDrehzVent1	:= 30.0;
				SollDrehzVent2	:= 30.0;

				IF (IstDrehzahlVent1 = SollDrehzVent1) THEN
					FreigabeVent1	:= FALSE;
				END_IF

				IF (IstDrehzahlVent2 = SollDrehzVent2) THEN
					FreigabeVent2	:= FALSE;
				END_IF

				// *** State exit ***
				IF (Tarifabschaltung) THEN
					stateEntry	:= TRUE;
					nextStep	:= TARIFABSCHALTUNG_FBTROCK;
				ELSIF (AnfVent1 OR AnfVent2)  THEN
					stateEntry	:= TRUE;
					nextStep	:= WARTEN_FBTROCK;
				ELSIF (FreigabeKlappen AND NOT FreigabeVent1 AND NOT FreigabeVent2) THEN
					stateEntry	:= TRUE;
					nextStep	:= KLAPPEN_ZU_FBTROCK;
				ELSIF (NOT FreigabeVent1 AND NOT FreigabeVent2) THEN
					stateEntry	:= TRUE;
					nextStep	:= WARTEN_FBTROCK;
				ELSE
					nextStep	:= curStep;
				END_IF

			//******************************************************************************************************************************************************************************************************************
			KLAPPEN_AUF_FBTROCK:

				//*** state entry ***
				IF (stateEntry) THEN
					stateEntry := FALSE;
				END_IF

				// *** State during	***
				SollDrehzVent1	:= 30.0;
				SollDrehzVent2	:= 30.0;

				IF (IstDrehzahlVent1 = SollDrehzVent1) THEN
					FreigabeVent1	:= FALSE;
				END_IF

				IF (IstDrehzahlVent2 = SollDrehzVent2) THEN
					FreigabeVent2	:= FALSE;
				END_IF

				TON_LaufzeitKlappen.IN	:= NOT FreigabeVent1 AND NOT FreigabeVent2;
				TON_LaufzeitKlappen.PT	:= UDINT_TO_TIME(LaufzeitKlappen);

				FreigabeKlappen			:= TON_LaufzeitKlappen.IN;

				// *** State exit ***
				IF (Tarifabschaltung) THEN
					stateEntry				:= TRUE;
					TON_LaufzeitKlappen.IN	:= FALSE;
					nextStep				:= TARIFABSCHALTUNG_FBTROCK;
				ELSIF (NOT AnfLuftentf) OR (NOT (AnfVent1 OR AnfVent2)) THEN
					stateEntry				:= TRUE;
					TON_LaufzeitKlappen.IN	:= FALSE;
					nextStep				:= KLAPPEN_ZU_FBTROCK;
				ELSIF (TON_LaufzeitKlappen.Q) THEN
					stateEntry				:= TRUE;
					TON_LaufzeitKlappen.IN	:= FALSE;
					nextStep				:= LA_EIN_VORBEREITUNG_FBTROCK;
				ELSE
					nextStep				:= curStep;
				END_IF

			//******************************************************************************************************************************************************************************************************************
			KLAPPEN_ZU_FBTROCK:

				//*** state entry ***
				IF (stateEntry) THEN
					stateEntry := FALSE;
				END_IF

				// *** State during	***
				SollDrehzVent1	:= 30.0;
				SollDrehzVent2	:= 30.0;

				IF (IstDrehzahlVent1 = SollDrehzVent1) THEN
					FreigabeVent1	:= FALSE;
				END_IF

				IF (IstDrehzahlVent2 = SollDrehzVent2) THEN
					FreigabeVent2	:= FALSE;
				END_IF

				TON_LaufzeitKlappen.IN	:= NOT FreigabeVent1 AND NOT FreigabeVent2;
				TON_LaufzeitKlappen.PT	:= UDINT_TO_TIME(LaufzeitKlappen);

				FreigabeKlappen			:= NOT TON_LaufzeitKlappen.IN;

				// *** State exit ***
				IF (Tarifabschaltung) THEN
					stateEntry				:= TRUE;
					TON_LaufzeitKlappen.IN	:= FALSE;
					nextStep				:= TARIFABSCHALTUNG_FBTROCK;
				ELSIF (AnfLuftentf) THEN
					stateEntry				:= TRUE;
					TON_LaufzeitKlappen.IN	:= FALSE;
					nextStep				:= KLAPPEN_AUF_FBTROCK;
				ELSIF (TON_LaufzeitKlappen.Q) AND (AnfVent1 OR AnfVent2) THEN
					stateEntry				:= TRUE;
					TON_LaufzeitKlappen.IN	:= FALSE;
					nextStep				:= VENT_EIN_FBTROCK;
				ELSIF (TON_LaufzeitKlappen.Q AND NOT AnfVent1 AND NOT AnfVent2) THEN
					stateEntry				:= TRUE;
					TON_LaufzeitKlappen.IN	:= FALSE;
					nextStep				:= WARTEN_FBTROCK;
				ELSE
					nextStep				:= curStep;
				END_IF

			//******************************************************************************************************************************************************************************************************************
			LA_EIN_VORBEREITUNG_FBTROCK:

				//*** state entry ***
				IF (stateEntry) THEN
					stateEntry := FALSE;
				END_IF

				// *** State during	***
				TON_AnlaufverzVent2.IN		:= FreigabeVent1;
				TON_AnlaufverzVent2.PT		:= UDINT_TO_TIME(AnlaufverzVent2);

				TON_LuftentfVorbereitung.IN	:= FreigabeVent1;
				TON_LuftentfVorbereitung.PT	:= UDINT_TO_TIME(EinschaltverzLuftentf);

				FreigabeVent1			:= TRUE;
				FreigabeVent2			:= AnfVent2 AND (TON_AnlaufverzVent2.Q);

				IF (Strombegrenzung AND (DrehzahlVent1Leistung >= DrehzahlBeiStrombegrenzung)) THEN
					SollDrehzVent1			:= DrehzahlBeiStrombegrenzung;
					SollDrehzVent2			:= DrehzahlBeiStrombegrenzung;
				ELSE
					SollDrehzVent1			:= DrehzahlVent1Leistung;
					SollDrehzVent2			:= DrehzahlVent2Leistung;
				END_IF

				// *** State exit ***
				IF (Tarifabschaltung) THEN
					stateEntry					:= TRUE;
					TON_LuftentfVorbereitung.IN	:= FALSE;
					nextStep					:= TARIFABSCHALTUNG_FBTROCK;
				ELSIF (NOT AnfLuftentf) THEN
					stateEntry					:= TRUE;
					TON_LuftentfVorbereitung.IN	:= FALSE;
					nextStep					:= KLAPPEN_ZU_FBTROCK;
				ELSIF (TON_LuftentfVorbereitung.Q) THEN
					stateEntry					:= TRUE;
					TON_LuftentfVorbereitung.IN	:= FALSE;
					nextStep					:= LA_EIN_FBTROCK;
				ELSE
					nextStep	:= curStep;
				END_IF

			//******************************************************************************************************************************************************************************************************************
			LA_EIN_FBTROCK:

				//*** state entry ***
				IF (stateEntry) THEN
					stateEntry := FALSE;
				END_IF

				// *** State during	***
				FreigabeLuftentf	:= TRUE;

				// *** State exit ***
				nextStep			:= VENT_EIN_FBTROCK;

			//******************************************************************************************************************************************************************************************************************
			LA_AUS_VORBEREITUNG_FBTROCK:

				//*** state entry ***
				IF (stateEntry) THEN
					stateEntry := FALSE;
				END_IF

				// *** State during	***
				TON_AuslaufzeitLuftentf.IN	:= NOT KeineKlappenAmLuftentf;
				TON_AuslaufzeitLuftentf.PT	:= UDINT_TO_TIME(AuslaufzeitLuftentfeuchter);

				FreigabeLuftentf			:= FALSE;

				IF (Strombegrenzung AND (DrehzahlVent1Leistung >= DrehzahlBeiStrombegrenzung)) THEN
					SollDrehzVent1			:= DrehzahlBeiStrombegrenzung;
					SollDrehzVent2			:= DrehzahlBeiStrombegrenzung;
				ELSE
					SollDrehzVent1			:= DrehzahlVent1Leistung;
					SollDrehzVent2			:= DrehzahlVent2Leistung;
				END_IF

				// *** State exit ***
				IF (Tarifabschaltung AND NOT BetriebsmldgLuftentf) THEN
					stateEntry					:= TRUE;
					TON_AuslaufzeitLuftentf.IN	:= FALSE;
					nextStep					:= TARIFABSCHALTUNG_FBTROCK;
				ELSIF (NOT AnfVent1 AND NOT AnfVent2 AND NOT BetriebsmldgLuftentf) THEN
					stateEntry					:= TRUE;
					TON_AuslaufzeitLuftentf.IN	:= FALSE;
					nextStep					:= VENT_AUS_FBTROCK;
				ELSIF (AnfLuftentf) THEN
					stateEntry					:= TRUE;
					TON_AuslaufzeitLuftentf.IN	:= FALSE;
					nextStep					:= LA_EIN_FBTROCK;
				ELSIF ((TON_AuslaufzeitLuftentf.Q OR KeineKlappenAmLuftentf) AND NOT BetriebsmldgLuftentf) THEN
					stateEntry					:= TRUE;
					TON_AuslaufzeitLuftentf.IN	:= FALSE;
					nextStep					:= MESSUNG_FBTROCK;
				ELSE
					nextStep					:= curStep;
				END_IF

			//******************************************************************************************************************************************************************************************************************
			MESSUNG_FBTROCK:

				//*** state entry ***
				IF (stateEntry) THEN
					stateEntry := FALSE;
				END_IF

				// *** State during	***
				TON_AnlaufverzVent2.IN	:= FreigabeVent1;
				TON_AnlaufverzVent2.PT	:= UDINT_TO_TIME(AnlaufverzVent2);

				FreigabeVent1			:= TRUE;
				FreigabeVent2			:= AnfVent2 AND (TON_AnlaufverzVent2.Q);

				IF (Strombegrenzung AND (DrehzahlVent1Leistung >= DrehzahlBeiStrombegrenzung)) THEN
					SollDrehzVent1			:= DrehzahlBeiStrombegrenzung;
					SollDrehzVent2			:= DrehzahlBeiStrombegrenzung;
				ELSE
					SollDrehzVent1			:= DrehzahlVent1Max;
					IF (IstDrehzahlVent1 = SollDrehzVent1) THEN
						SollDrehzVent2			:= DrehzahlVent2Max;
					END_IF
				END_IF

				TON_Messung.IN		:= (IstDrehzahlVent1 = DrehzahlVent1Max) AND ((IstDrehzahlVent2 = DrehzahlVent2Max) OR (NOT AnfVent2));
				TON_Messung.PT		:= UDINT_TO_TIME(MessdauerLuftgeschw);
				MessungAktiv		:= TON_Messung.IN;

				// *** State exit ***
				IF (Tarifabschaltung) THEN
					stateEntry					:= TRUE;
					MessungAktiv				:= FALSE;
					TON_Messung.IN				:= FALSE;
					TON_AnlaufverzVent2.IN		:= FALSE;
					nextStep					:= TARIFABSCHALTUNG_FBTROCK;
				ELSIF (NOT AnfVent1 AND NOT AnfVent2) THEN
					stateEntry					:= TRUE;
					MessungAktiv				:= FALSE;
					TON_Messung.IN				:= FALSE;
					TON_AnlaufverzVent2.IN		:= FALSE;
					nextStep					:= VENT_AUS_FBTROCK;
				ELSIF (TON_Messung.Q OR Strombegrenzung OR KeineKlappenAmLuftentf) THEN
					IF (NOT Strombegrenzung) THEN
						IF (AnfVent1 AND NOT AnfVent2) AND TON_Messung.Q THEN
							LuftgeschwBeiMaxDrehzahl1Vent	:= Mittelwertbildung.y;
						ELSIF (TON_Messung.Q) THEN
							LuftgeschwBeiMaxDrehzahl2Vent	:= Mittelwertbildung.y;
						END_IF
					END_IF
					stateEntry					:= TRUE;
					MessungAktiv				:= FALSE;
					TON_Messung.IN				:= FALSE;
					TON_AnlaufverzVent2.IN		:= FALSE;
					nextStep					:= KLAPPEN_ZU_FBTROCK;
				ELSIF (AnfLuftentf) THEN
					stateEntry					:= TRUE;
					MessungAktiv				:= FALSE;
					TON_Messung.IN				:= FALSE;
					TON_AnlaufverzVent2.IN		:= FALSE;
					nextStep					:= LA_EIN_FBTROCK;
				ELSE
					nextStep					:= curStep;
				END_IF

			//******************************************************************************************************************************************************************************************************************
			TARIFABSCHALTUNG_FBTROCK:

				//*** state entry ***
				IF (stateEntry) THEN
					stateEntry := FALSE;
				END_IF

				// *** State during	***
				SollDrehzVent1	:= 30.0;
				SollDrehzVent2	:= 30.0;

				FreigabeLuftentf		:= FALSE;

				IF (IstDrehzahlVent1 = SollDrehzVent1) THEN
					FreigabeVent1		:= FALSE;
				END_IF

				IF (IstDrehzahlVent2 = SollDrehzVent2) THEN
					FreigabeVent2		:= FALSE;
				END_IF

				FreigabeKlappen			:= FreigabeVent1 OR FreigabeVent2;

				// *** State exit ***
				IF (NOT Tarifabschaltung) THEN
					stateEntry	:= TRUE;
					nextStep	:= WARTEN_FBTROCK;
				ELSE
					nextStep	:= curStep;
				END_IF

		END_CASE

		//Mittelwert Luftmenge berechnen
		IF (sekTick AND MessungAktiv) THEN
			Mittelwertbildung.enable	:= MessungAktiv;
			Mittelwertbildung.x			:= LuftgeschwAktuell;
			Mittelwertbildung.base		:= 30;
			Mittelwertbildung();
		END_IF

		//Funktionsblöcke aufrufen
		TON_AnlaufverzVent2();
		TON_AuslaufzeitLuftentf();
		TON_LaufzeitKlappen();
		TON_LuftentfVorbereitung();
		TON_Messung();

	ELSE

		FreigabeKlappen				:= FALSE;
		FreigabeLuftentf			:= FALSE;
		FreigabeVent1				:= FALSE;
		FreigabeVent2				:= FALSE;
		MessungAktiv				:= FALSE;
		SollDrehzVent1				:= 0.0;
		SollDrehzVent2				:= 0.0;
		TON_AnlaufverzVent2.IN		:= FALSE;
		TON_AuslaufzeitLuftentf.IN	:= FALSE;
		TON_LaufzeitKlappen.IN		:= FALSE;
		TON_Messung.IN				:= FALSE;
		TON_LuftentfVorbereitung.IN	:= FALSE;
		curStep						:= WARTEN_FBTROCK;
		nextStep					:= WARTEN_FBTROCK;

	END_IF

END_FUNCTION_BLOCK
```
